LIN {X 0,Y 222.683,Z 907.794,A -85,B 0,C 180,E1 -20580.36,E2 -20580.36} C_VEL
LIN {X 0,Y 221.967,Z 912.88,A -85,B 0,C 180,E1 -20581.113,E2 -20581.113} C_VEL
LIN {X 0,Y 221.213,Z 924.782,A -85,B 0,C 180,E1 -20583.298,E2 -20583.298} C_VEL
LIN {X 0,Y 220.004,Z 934.618,A -85,B 0,C 180,E1 -20585.467,E2 -20585.467} C_VEL
LIN {X 0,Y 218.54,Z 943.393,A -85,B 0,C 180,E1 -20587.802,E2 -20587.802} C_VEL
LIN {X 0,Y 216.195,Z 951.788,A -85,B 0,C 180,E1 -20590.515,E2 -20590.515} C_VEL
LIN {X 0,Y 214.636,Z 957.677,A -85,B 0,C 180,E1 -20592.865,E2 -20592.865} C_VEL
LIN {X 0,Y 213.497,Z 963.435,A -85,B 0,C 180,E1 -20595.71,E2 -20595.71} C_VEL
LIN {X 0,Y 212.841,Z 968.001,A -85,B 0,C 180,E1 -20598.577,E2 -20598.577} C_VEL
LIN {X 0,Y 212.752,Z 972.374,A -85,B 0,C 180,E1 -20602.314,E2 -20602.314} C_VEL
LIN {X 0,Y 212.967,Z 973.999,A -85,B 0,C 180,E1 -20604.322,E2 -20604.322} C_VEL
LIN {X 0,Y 213.246,Z 975.11,A -85,B 0,C 180,E1 -20606.224,E2 -20606.224} C_VEL
LIN {X 0,Y 213.487,Z 975.797,A -85,B 0,C 180,E1 -20608.117,E2 -20608.117} C_VEL
LIN {X 0,Y 213.744,Z 976.061,A -85,B 0,C 180,E1 -20610.003,E2 -20610.003} C_VEL
LIN {X 0,Y 213.491,Z 975.785,A -85,B 0,C 180,E1 -20611.89,E2 -20611.89} C_VEL
LIN {X 0,Y 213.259,Z 975.091,A -85,B 0,C 180,E1 -20613.782,E2 -20613.782} C_VEL
LIN {X 0,Y 212.992,Z 973.972,A -85,B 0,C 180,E1 -20615.684,E2 -20615.684} C_VEL
LIN {X 0,Y 212.76,Z 972.318,A -85,B 0,C 180,E1 -20617.703,E2 -20617.703} C_VEL
LIN {X 0,Y 212.843,Z 968.742,A -85,B 0,C 180,E1 -20620.948,E2 -20620.948} C_VEL
LIN {X 0,Y 213.212,Z 967.284,A -85,B 0,C 180,E1 -20623.344,E2 -20623.344} C_VEL
LIN {X 0,Y 214.757,Z 963.862,A -85,B 0,C 180,E1 -20627.132,E2 -20627.132} C_VEL
LIN {X 0,Y 217.509,Z 959.058,A -85,B 0,C 180,E1 -20630.823,E2 -20630.823} C_VEL
LIN {X 0,Y 221.527,Z 952.942,A -85,B 0,C 180,E1 -20634.361,E2 -20634.361} C_VEL
LIN {X 0,Y 224.855,Z 947.353,A -85,B 0,C 180,E1 -20636.953,E2 -20636.953} C_VEL
LIN {X 0,Y 229.122,Z 939.872,A -85,B 0,C 180,E1 -20639.9,E2 -20639.9} C_VEL
LIN {X 0,Y 234.33,Z 930.73,A -85,B 0,C 180,E1 -20642.884,E2 -20642.884} C_VEL
LIN {X 0,Y 239.363,Z 919.685,A -85,B 0,C 180,E1 -20646.344,E2 -20646.344} C_VEL
LIN {X 0,Y 243.363,Z 909.541,A -85,B 0,C 180,E1 -20649.448,E2 -20649.448} C_VEL
LIN {X 0,Y 247.656,Z 898.848,A -85,B 0,C 180,E1 -20652.931,E2 -20652.931} C_VEL
LIN {X 0,Y 249.749,Z 893.918,A -85,B 0,C 180,E1 -20654.712,E2 -20654.712} C_VEL
LIN {X 0,Y 250.439,Z 892.26,A -85,B 0,C 180,E1 -20655.447,E2 -20655.447} C_VEL
LIN {X 0,Y 251.117,Z 890.281,A -85,B 0,C 180,E1 -20656.694,E2 -20656.694} C_VEL
LIN {X 0,Y 251.911,Z 888.053,A -85,B 0,C 180,E1 -20658.877,E2 -20658.877} C_VEL
LIN {X 0,Y 252.305,Z 887.295,A -85,B 0,C 180,E1 -20660.158,E2 -20660.158} C_VEL
LIN {X 0,Y 252.805,Z 886.985,A -85,B 0,C 180,E1 -20662.295,E2 -20662.295} C_VEL
LIN {X 0,Y 253.061,Z 887.829,A -85,B 0,C 180,E1 -20664.323,E2 -20664.323} C_VEL
LIN {X 0,Y 252.783,Z 889.741,A -85,B 0,C 180,E1 -20666.523,E2 -20666.523} C_VEL
LIN {X 0,Y 251.661,Z 893.245,A -85,B 0,C 180,E1 -20668.893,E2 -20668.893} C_VEL
LIN {X 0,Y 250.434,Z 895.146,A -85,B 0,C 180,E1 -20669.659,E2 -20669.659} C_VEL
LIN {X 0,Y 243.614,Z 903.148,A -85,B 0,C 180,E1 -20672.511,E2 -20672.511} C_VEL
LIN {X 0,Y 237.346,Z 909.214,A -85,B 0,C 180,E1 -20675.509,E2 -20675.509} C_VEL
LIN {X 0,Y 233.205,Z 912.764,A -85,B 0,C 180,E1 -20677.87,E2 -20677.87} C_VEL
LIN {X 0,Y 227.046,Z 916.649,A -85,B 0,C 180,E1 -20681.968,E2 -20681.968} C_VEL
LIN {X 0,Y 222.953,Z 918.003,A -85,B 0,C 180,E1 -20685.394,E2 -20685.394} C_VEL
LIN {X 0,Y 219.57,Z 918.045,A -85,B 0,C 180,E1 -20688.928,E2 -20688.928} C_VEL
LIN {X 0,Y 217.142,Z 916.466,A -85,B 0,C 180,E1 -20692.561,E2 -20692.561} C_VEL
LIN {X 0,Y 215.54,Z 913.407,A -85,B 0,C 180,E1 -20696.261,E2 -20696.261} C_VEL
LIN {X 0,Y 214.542,Z 910.085,A -85,B 0,C 180,E1 -20699.062,E2 -20699.062} C_VEL
LIN {X 0,Y 214.067,Z 905.794,A -85,B 0,C 180,E1 -20701.882,E2 -20701.882} C_VEL
LIN {X 0,Y 213.844,Z 899.385,A -85,B 0,C 180,E1 -20705.186,E2 -20705.186} C_VEL
LIN {X 0,Y 214.309,Z 892.64,A -85,B 0,C 180,E1 -20708.012,E2 -20708.012} C_VEL
LIN {X 0,Y 214.845,Z 884.897,A -85,B 0,C 180,E1 -20710.746,E2 -20710.746} C_VEL
LIN {X 0,Y 215.793,Z 874.678,A -85,B 0,C 180,E1 -20713.658,E2 -20713.658} C_VEL
LIN {X 0,Y 216.972,Z 862.599,A -85,B 0,C 180,E1 -20716.465,E2 -20716.465} C_VEL
LIN {X 0,Y 218.067,Z 851.603,A -85,B 0,C 180,E1 -20718.558,E2 -20718.558} C_VEL
LIN {X 0,Y 218.521,Z 845.919,A -85,B 0,C 180,E1 -20719.493,E2 -20719.493} C_VEL
LIN {X 0,Y 215.547,Z 833.553,A -85,B 0,C 180,E1 -20721.358,E2 -20721.358} C_VEL
LIN {X 0,Y 213.843,Z 825.837,A -85,B 0,C 180,E1 -20722.392,E2 -20722.392} C_VEL
LIN {X 0,Y 213.775,Z 825.841,A -85,B 0,C 180,E1 -20727.416,E2 -20727.416} C_VEL
LIN {X 0,Y 213.767,Z 825.845,A -85,B 0,C 180,E1 -20731.738,E2 -20731.738} C_VEL
LIN {X 0,Y 213.75,Z 825.853,A -85,B 0,C 180,E1 -20736.287,E2 -20736.287} C_VEL
LIN {X 0,Y 213.706,Z 825.861,A -85,B 0,C 180,E1 -20741.127,E2 -20741.127} C_VEL
LIN {X 0,Y 213.709,Z 825.861,A -85,B 0,C 180,E1 -20743.678,E2 -20743.678} C_VEL
LIN {X 0,Y 213.708,Z 825.858,A -85,B 0,C 180,E1 -20746.344,E2 -20746.344} C_VEL
LIN {X 0,Y 213.711,Z 825.865,A -85,B 0,C 180,E1 -20751.327,E2 -20751.327} C_VEL
LIN {X 0,Y 213.774,Z 825.945,A -85,B 0,C 180,E1 -20755.566,E2 -20755.566} C_VEL
LIN {X 0,Y 214.833,Z 828.734,A -85,B 0,C 180,E1 -20756.044,E2 -20756.044} C_VEL
LIN {X 0,Y 219.16,Z 837.219,A -85,B 0,C 180,E1 -20757.82,E2 -20757.82} C_VEL
LIN {X 0,Y 223.302,Z 847.04,A -85,B 0,C 180,E1 -20759.94,E2 -20759.94} C_VEL
LIN {X 0,Y 226.253,Z 856.184,A -85,B 0,C 180,E1 -20762.01,E2 -20762.01} C_VEL
LIN {X 0,Y 228.469,Z 865.319,A -85,B 0,C 180,E1 -20764.25,E2 -20764.25} C_VEL
LIN {X 0,Y 228.457,Z 867.41,A -85,B 0,C 180,E1 -20764.73,E2 -20764.73} C_VEL
LIN {X 0,Y 226.319,Z 876.166,A -85,B 0,C 180,E1 -20766.673,E2 -20766.673} C_VEL
LIN {X 0,Y 224.064,Z 884.201,A -85,B 0,C 180,E1 -20768.853,E2 -20768.853} C_VEL
LIN {X 0,Y 222.104,Z 890.846,A -85,B 0,C 180,E1 -20771.071,E2 -20771.071} C_VEL
LIN {X 0,Y 220.379,Z 896.376,A -85,B 0,C 180,E1 -20773.318,E2 -20773.318} C_VEL
LIN {X 0,Y 218.689,Z 901.747,A -85,B 0,C 180,E1 -20776.05,E2 -20776.05} C_VEL
LIN {X 0,Y 216.938,Z 906.012,A -85,B 0,C 180,E1 -20778.788,E2 -20778.788} C_VEL
LIN {X 0,Y 216.156,Z 908.239,A -85,B 0,C 180,E1 -20780.641,E2 -20780.641} C_VEL
LIN {X 0,Y 215.625,Z 910.035,A -85,B 0,C 180,E1 -20782.506,E2 -20782.506} C_VEL
LIN {X 0,Y 215.277,Z 911.377,A -85,B 0,C 180,E1 -20784.376,E2 -20784.376} C_VEL
LIN {X 0,Y 214.632,Z 912.955,A -85,B 0,C 180,E1 -20788.12,E2 -20788.12} C_VEL
LIN {X 0,Y 214.545,Z 913.183,A -85,B 0,C 180,E1 -20789.997,E2 -20789.997} C_VEL
LIN {X 0,Y 214.897,Z 912.41,A -85,B 0,C 180,E1 -20793.747,E2 -20793.747} C_VEL
LIN {X 0,Y 215.247,Z 911.466,A -85,B 0,C 180,E1 -20795.618,E2 -20795.618} C_VEL
LIN {X 0,Y 215.52,Z 910.172,A -85,B 0,C 180,E1 -20797.491,E2 -20797.491} C_VEL
LIN {X 0,Y 216.517,Z 907.366,A -85,B 0,C 180,E1 -20800.28,E2 -20800.28} C_VEL
LIN {X 0,Y 218.106,Z 903.519,A -85,B 0,C 180,E1 -20803.032,E2 -20803.032} C_VEL
LIN {X 0,Y 219.788,Z 898.601,A -85,B 0,C 180,E1 -20805.768,E2 -20805.768} C_VEL
LIN {X 0,Y 221.653,Z 892.417,A -85,B 0,C 180,E1 -20808.482,E2 -20808.482} C_VEL
LIN {X 0,Y 224.005,Z 884.641,A -85,B 0,C 180,E1 -20811.146,E2 -20811.146} C_VEL
LIN {X 0,Y 226.211,Z 876.701,A -85,B 0,C 180,E1 -20813.332,E2 -20813.332} C_VEL
LIN {X 0,Y 228.66,Z 866.99,A -85,B 0,C 180,E1 -20815.483,E2 -20815.483} C_VEL
LIN {X 0,Y 228.253,Z 863.798,A -85,B 0,C 180,E1 -20816.264,E2 -20816.264} C_VEL
LIN {X 0,Y 225.979,Z 855.105,A -85,B 0,C 180,E1 -20818.384,E2 -20818.384} C_VEL
LIN {X 0,Y 223.287,Z 846.892,A -85,B 0,C 180,E1 -20820.234,E2 -20820.234} C_VEL
LIN {X 0,Y 218.787,Z 836.479,A -85,B 0,C 180,E1 -20822.493,E2 -20822.493} C_VEL
LIN {X 0,Y 214.007,Z 826.929,A -85,B 0,C 180,E1 -20824.448,E2 -20824.448} C_VEL
LIN {X 0,Y 213.782,Z 825.857,A -85,B 0,C 180,E1 -20824.636,E2 -20824.636} C_VEL
LIN {X 0,Y 213.777,Z 825.858,A -85,B 0,C 180,E1 -20828.65,E2 -20828.65} C_VEL
LIN {X 0,Y 213.817,Z 825.851,A -85,B 0,C 180,E1 -20831.096,E2 -20831.096} C_VEL
LIN {X 0,Y 213.828,Z 825.851,A -85,B 0,C 180,E1 -20833.69,E2 -20833.69} C_VEL
LIN {X 0,Y 213.831,Z 825.846,A -85,B 0,C 180,E1 -20836.353,E2 -20836.353} C_VEL
LIN {X 0,Y 213.821,Z 825.851,A -85,B 0,C 180,E1 -20839.105,E2 -20839.105} C_VEL
LIN {X 0,Y 213.749,Z 825.859,A -85,B 0,C 180,E1 -20843.712,E2 -20843.712} C_VEL
LIN {X 0,Y 213.784,Z 825.851,A -85,B 0,C 180,E1 -20848.722,E2 -20848.722} C_VEL
LIN {X 0,Y 213.813,Z 825.852,A -85,B 0,C 180,E1 -20852.601,E2 -20852.601} C_VEL
LIN {X 0,Y 213.839,Z 825.85,A -85,B 0,C 180,E1 -20856.951,E2 -20856.951} C_VEL
LIN {X 0,Y 213.93,Z 825.834,A -85,B 0,C 180,E1 -20862.802,E2 -20862.802} C_VEL
LIN {X 0,Y 213.966,Z 825.83,A -85,B 0,C 180,E1 -20866.707,E2 -20866.707} C_VEL
LIN {X 0,Y 214.152,Z 825.8,A -85,B 0,C 180,E1 -20870.556,E2 -20870.556} C_VEL
LIN {X 0,Y 214.211,Z 825.802,A -85,B 0,C 180,E1 -20872.459,E2 -20872.459} C_VEL
LIN {X 0,Y 214.43,Z 825.773,A -85,B 0,C 180,E1 -20878.122,E2 -20878.122} C_VEL
LIN {X 0,Y 214.535,Z 825.767,A -85,B 0,C 180,E1 -20880,E2 -20880} C_VEL
LIN {X 0,Y 214.429,Z 825.78,A -85,B 0,C 180,E1 -20881.878,E2 -20881.878} C_VEL
LIN {X 0,Y 214.208,Z 825.805,A -85,B 0,C 180,E1 -20887.541,E2 -20887.541} C_VEL
LIN {X 0,Y 214.009,Z 825.822,A -85,B 0,C 180,E1 -20891.364,E2 -20891.364} C_VEL
LIN {X 0,Y 213.919,Z 825.84,A -85,B 0,C 180,E1 -20895.238,E2 -20895.238} C_VEL
LIN {X 0,Y 213.822,Z 825.853,A -85,B 0,C 180,E1 -20899.189,E2 -20899.189} C_VEL
LIN {X 0,Y 213.789,Z 825.855,A -85,B 0,C 180,E1 -20903.234,E2 -20903.234} C_VEL
LIN {X 0,Y 213.773,Z 825.851,A -85,B 0,C 180,E1 -20907.429,E2 -20907.429} C_VEL
LIN {X 0,Y 213.781,Z 826.027,A -85,B 0,C 180,E1 -20909.006,E2 -20909.006} C_VEL
LIN {X 0,Y 215.008,Z 831.466,A -85,B 0,C 180,E1 -20913.758,E2 -20913.758} C_VEL
LIN {X 0,Y 216.095,Z 836.967,A -85,B 0,C 180,E1 -20918.165,E2 -20918.165} C_VEL
LIN {X 0,Y 217.106,Z 842.018,A -85,B 0,C 180,E1 -20921.886,E2 -20921.886} C_VEL
LIN {X 0,Y 218.334,Z 848.445,A -85,B 0,C 180,E1 -20926.347,E2 -20926.347} C_VEL
LIN {X 0,Y 219.202,Z 854.278,A -85,B 0,C 180,E1 -20930.121,E2 -20930.121} C_VEL
LIN {X 0,Y 217.328,Z 861.535,A -85,B 0,C 180,E1 -20934.407,E2 -20934.407} C_VEL
LIN {X 0,Y 217.039,Z 862.617,A -85,B 0,C 180,E1 -20935.044,E2 -20935.044} C_VEL
LIN {X 0,Y 219.827,Z 877.43,A -85,B 0,C 180,E1 -20936.433,E2 -20936.433} C_VEL
LIN {X 0,Y 221.389,Z 890.305,A -85,B 0,C 180,E1 -20937.887,E2 -20937.887} C_VEL
LIN {X 0,Y 222.027,Z 903.006,A -85,B 0,C 180,E1 -20939.576,E2 -20939.576} C_VEL
LIN {X 0,Y 221.967,Z 912.88,A -85,B 0,C 180,E1 -20941.113,E2 -20941.113} C_VEL
LIN {X 0,Y 221.111,Z 917.912,A -85,B 0,C 180,E1 -20941.916,E2 -20941.916} C_VEL
LIN {X 0,Y 217.74,Z 925.844,A -85,B 0,C 180,E1 -20943.193,E2 -20943.193} C_VEL
LIN {X 0,Y 214.028,Z 933.31,A -85,B 0,C 180,E1 -20944.639,E2 -20944.639} C_VEL
LIN {X 0,Y 212.67,Z 937.55,A -85,B 0,C 180,E1 -20945.694,E2 -20945.694} C_VEL
LIN {X 0,Y 211.476,Z 943.865,A -85,B 0,C 180,E1 -20947.535,E2 -20947.535} C_VEL
LIN {X 0,Y 209.056,Z 952.07,A -85,B 0,C 180,E1 -20950.36,E2 -20950.36} C_VEL
LIN {X 0,Y 207.319,Z 958.712,A -85,B 0,C 180,E1 -20953.257,E2 -20953.257} C_VEL
LIN {X 0,Y 206.231,Z 964.049,A -85,B 0,C 180,E1 -20956.203,E2 -20956.203} C_VEL
LIN {X 0,Y 205.69,Z 968.251,A -85,B 0,C 180,E1 -20959.172,E2 -20959.172} C_VEL
LIN {X 0,Y 205.702,Z 971.488,A -85,B 0,C 180,E1 -20962.228,E2 -20962.228} C_VEL
LIN {X 0,Y 205.873,Z 972.952,A -85,B 0,C 180,E1 -20964.125,E2 -20964.125} C_VEL
LIN {X 0,Y 206.187,Z 974.072,A -85,B 0,C 180,E1 -20966.095,E2 -20966.095} C_VEL
LIN {X 0,Y 206.434,Z 974.761,A -85,B 0,C 180,E1 -20968.053,E2 -20968.053} C_VEL
LIN {X 0,Y 206.709,Z 975.028,A -85,B 0,C 180,E1 -20970.003,E2 -20970.003} C_VEL
LIN {X 0,Y 206.439,Z 974.749,A -85,B 0,C 180,E1 -20971.954,E2 -20971.954} C_VEL
LIN {X 0,Y 206.201,Z 974.052,A -85,B 0,C 180,E1 -20973.912,E2 -20973.912} C_VEL
LIN {X 0,Y 205.919,Z 972.928,A -85,B 0,C 180,E1 -20975.88,E2 -20975.88} C_VEL
LIN {X 0,Y 205.65,Z 970.404,A -85,B 0,C 180,E1 -20978.85,E2 -20978.85} C_VEL
LIN {X 0,Y 205.868,Z 967.591,A -85,B 0,C 180,E1 -20981.324,E2 -20981.324} C_VEL
LIN {X 0,Y 206.273,Z 966.276,A -85,B 0,C 180,E1 -20983.801,E2 -20983.801} C_VEL
LIN {X 0,Y 207.941,Z 963.094,A -85,B 0,C 180,E1 -20987.712,E2 -20987.712} C_VEL
LIN {X 0,Y 210.859,Z 958.713,A -85,B 0,C 180,E1 -20991.511,E2 -20991.511} C_VEL
LIN {X 0,Y 216.27,Z 951.338,A -85,B 0,C 180,E1 -20996.024,E2 -20996.024} C_VEL
LIN {X 0,Y 221.008,Z 943.837,A -85,B 0,C 180,E1 -20999.534,E2 -20999.534} C_VEL
LIN {X 0,Y 225.196,Z 937.404,A -85,B 0,C 180,E1 -21002.045,E2 -21002.045} C_VEL
LIN {X 0,Y 229.467,Z 930.54,A -85,B 0,C 180,E1 -21004.411,E2 -21004.411} C_VEL
LIN {X 0,Y 234.602,Z 920.476,A -85,B 0,C 180,E1 -21007.778,E2 -21007.778} C_VEL
LIN {X 0,Y 238.991,Z 911.214,A -85,B 0,C 180,E1 -21010.87,E2 -21010.87} C_VEL
LIN {X 0,Y 243.188,Z 902.406,A -85,B 0,C 180,E1 -21013.918,E2 -21013.918} C_VEL
LIN {X 0,Y 245.543,Z 897.892,A -85,B 0,C 180,E1 -21015.692,E2 -21015.692} C_VEL
LIN {X 0,Y 246.382,Z 895.927,A -85,B 0,C 180,E1 -21016.796,E2 -21016.796} C_VEL
LIN {X 0,Y 246.856,Z 894.714,A -85,B 0,C 180,E1 -21017.754,E2 -21017.754} C_VEL
LIN {X 0,Y 247.445,Z 893.378,A -85,B 0,C 180,E1 -21019.213,E2 -21019.213} C_VEL
LIN {X 0,Y 248.037,Z 892.425,A -85,B 0,C 180,E1 -21021.438,E2 -21021.438} C_VEL
LIN {X 0,Y 248.183,Z 892.641,A -85,B 0,C 180,E1 -21023.511,E2 -21023.511} C_VEL
LIN {X 0,Y 247.944,Z 893.919,A -85,B 0,C 180,E1 -21025.465,E2 -21025.465} C_VEL
LIN {X 0,Y 247.657,Z 894.867,A -85,B 0,C 180,E1 -21026.432,E2 -21026.432} C_VEL
LIN {X 0,Y 246.544,Z 897.179,A -85,B 0,C 180,E1 -21028.173,E2 -21028.173} C_VEL
LIN {X 0,Y 245.079,Z 899.036,A -85,B 0,C 180,E1 -21028.924,E2 -21028.924} C_VEL
LIN {X 0,Y 239.652,Z 904.776,A -85,B 0,C 180,E1 -21031.061,E2 -21031.061} C_VEL
LIN {X 0,Y 232.928,Z 910.767,A -85,B 0,C 180,E1 -21034.056,E2 -21034.056} C_VEL
LIN {X 0,Y 228.423,Z 914.285,A -85,B 0,C 180,E1 -21036.423,E2 -21036.423} C_VEL
LIN {X 0,Y 225.661,Z 916.099,A -85,B 0,C 180,E1 -21038.054,E2 -21038.054} C_VEL
LIN {X 0,Y 220.57,Z 918.549,A -85,B 0,C 180,E1 -21041.42,E2 -21041.42} C_VEL
LIN {X 0,Y 218.324,Z 919.318,A -85,B 0,C 180,E1 -21043.159,E2 -21043.159} C_VEL
LIN {X 0,Y 214.415,Z 919.665,A -85,B 0,C 180,E1 -21046.736,E2 -21046.736} C_VEL
LIN {X 0,Y 212.716,Z 919.295,A -85,B 0,C 180,E1 -21048.566,E2 -21048.566} C_VEL
LIN {X 0,Y 210.19,Z 917.429,A -85,B 0,C 180,E1 -21052.314,E2 -21052.314} C_VEL
LIN {X 0,Y 208.477,Z 913.961,A -85,B 0,C 180,E1 -21056.134,E2 -21056.134} C_VEL
LIN {X 0,Y 207.445,Z 910.398,A -85,B 0,C 180,E1 -21059.029,E2 -21059.029} C_VEL
LIN {X 0,Y 206.964,Z 905.852,A -85,B 0,C 180,E1 -21061.946,E2 -21061.946} C_VEL
LIN {X 0,Y 206.738,Z 900.23,A -85,B 0,C 180,E1 -21064.875,E2 -21064.875} C_VEL
LIN {X 0,Y 207.156,Z 893.416,A -85,B 0,C 180,E1 -21067.799,E2 -21067.799} C_VEL
LIN {X 0,Y 207.657,Z 886.611,A -85,B 0,C 180,E1 -21070.291,E2 -21070.291} C_VEL
LIN {X 0,Y 208.354,Z 878.805,A -85,B 0,C 180,E1 -21072.665,E2 -21072.665} C_VEL
LIN {X 0,Y 209.142,Z 870.512,A -85,B 0,C 180,E1 -21074.847,E2 -21074.847} C_VEL
LIN {X 0,Y 209.99,Z 861.955,A -85,B 0,C 180,E1 -21076.778,E2 -21076.778} C_VEL
LIN {X 0,Y 211.155,Z 850.698,A -85,B 0,C 180,E1 -21078.936,E2 -21078.936} C_VEL
LIN {X 0,Y 211.291,Z 846.213,A -85,B 0,C 180,E1 -21079.687,E2 -21079.687} C_VEL
LIN {X 0,Y 208.404,Z 834.211,A -85,B 0,C 180,E1 -21081.54,E2 -21081.54} C_VEL
LIN {X 0,Y 206.788,Z 826.717,A -85,B 0,C 180,E1 -21082.571,E2 -21082.571} C_VEL
LIN {X 0,Y 206.704,Z 826.722,A -85,B 0,C 180,E1 -21087.865,E2 -21087.865} C_VEL
LIN {X 0,Y 206.717,Z 826.723,A -85,B 0,C 180,E1 -21091.788,E2 -21091.788} C_VEL
LIN {X 0,Y 206.708,Z 826.733,A -85,B 0,C 180,E1 -21095.31,E2 -21095.31} C_VEL
LIN {X 0,Y 206.655,Z 826.742,A -85,B 0,C 180,E1 -21100.253,E2 -21100.253} C_VEL
LIN {X 0,Y 206.637,Z 826.746,A -85,B 0,C 180,E1 -21104.415,E2 -21104.415} C_VEL
LIN {X 0,Y 206.637,Z 826.746,A -85,B 0,C 180,E1 -21108.439,E2 -21108.439} C_VEL
LIN {X 0,Y 206.698,Z 826.733,A -85,B 0,C 180,E1 -21113.483,E2 -21113.483} C_VEL
LIN {X 0,Y 206.736,Z 826.85,A -85,B 0,C 180,E1 -21114.18,E2 -21114.18} C_VEL
LIN {X 0,Y 207.778,Z 829.656,A -85,B 0,C 180,E1 -21114.689,E2 -21114.689} C_VEL
LIN {X 0,Y 212.372,Z 838.462,A -85,B 0,C 180,E1 -21116.667,E2 -21116.667} C_VEL
LIN {X 0,Y 216.471,Z 848.029,A -85,B 0,C 180,E1 -21118.858,E2 -21118.858} C_VEL
LIN {X 0,Y 219.657,Z 857.627,A -85,B 0,C 180,E1 -21121.156,E2 -21121.156} C_VEL
LIN {X 0,Y 221.764,Z 866.251,A -85,B 0,C 180,E1 -21123.373,E2 -21123.373} C_VEL
LIN {X 0,Y 222.115,Z 868.447,A -85,B 0,C 180,E1 -21123.955,E2 -21123.955} C_VEL
LIN {X 0,Y 219.887,Z 877.2,A -85,B 0,C 180,E1 -21125.948,E2 -21125.948} C_VEL
LIN {X 0,Y 217.527,Z 885.234,A -85,B 0,C 180,E1 -21128.186,E2 -21128.186} C_VEL
LIN {X 0,Y 215.47,Z 891.879,A -85,B 0,C 180,E1 -21130.465,E2 -21130.465} C_VEL
LIN {X 0,Y 213.659,Z 897.409,A -85,B 0,C 180,E1 -21132.777,E2 -21132.777} C_VEL
LIN {X 0,Y 211.88,Z 902.78,A -85,B 0,C 180,E1 -21135.592,E2 -21135.592} C_VEL
LIN {X 0,Y 210.053,Z 907.044,A -85,B 0,C 180,E1 -21138.416,E2 -21138.416} C_VEL
LIN {X 0,Y 209.228,Z 909.271,A -85,B 0,C 180,E1 -21140.328,E2 -21140.328} C_VEL
LIN {X 0,Y 208.673,Z 911.066,A -85,B 0,C 180,E1 -21142.254,E2 -21142.254} C_VEL
LIN {X 0,Y 208.291,Z 912.408,A -85,B 0,C 180,E1 -21144.187,E2 -21144.187} C_VEL
LIN {X 0,Y 207.612,Z 913.986,A -85,B 0,C 180,E1 -21148.057,E2 -21148.057} C_VEL
LIN {X 0,Y 207.521,Z 914.214,A -85,B 0,C 180,E1 -21149.997,E2 -21149.997} C_VEL
LIN {X 0,Y 207.888,Z 913.441,A -85,B 0,C 180,E1 -21153.873,E2 -21153.873} C_VEL
LIN {X 0,Y 208.258,Z 912.496,A -85,B 0,C 180,E1 -21155.807,E2 -21155.807} C_VEL
LIN {X 0,Y 208.581,Z 911.199,A -85,B 0,C 180,E1 -21157.742,E2 -21157.742} C_VEL
LIN {X 0,Y 209.609,Z 908.397,A -85,B 0,C 180,E1 -21160.623,E2 -21160.623} C_VEL
LIN {X 0,Y 211.267,Z 904.549,A -85,B 0,C 180,E1 -21163.462,E2 -21163.462} C_VEL
LIN {X 0,Y 213.036,Z 899.631,A -85,B 0,C 180,E1 -21166.281,E2 -21166.281} C_VEL
LIN {X 0,Y 215.009,Z 893.445,A -85,B 0,C 180,E1 -21169.075,E2 -21169.075} C_VEL
LIN {X 0,Y 217.469,Z 885.67,A -85,B 0,C 180,E1 -21171.813,E2 -21171.813} C_VEL
LIN {X 0,Y 219.779,Z 877.73,A -85,B 0,C 180,E1 -21174.057,E2 -21174.057} C_VEL
LIN {X 0,Y 222.226,Z 868.036,A -85,B 0,C 180,E1 -21176.276,E2 -21176.276} C_VEL
LIN {X 0,Y 220.133,Z 859.17,A -85,B 0,C 180,E1 -21178.609,E2 -21178.609} C_VEL
LIN {X 0,Y 217.112,Z 849.564,A -85,B 0,C 180,E1 -21180.929,E2 -21180.929} C_VEL
LIN {X 0,Y 212.971,Z 839.724,A -85,B 0,C 180,E1 -21183.205,E2 -21183.205} C_VEL
LIN {X 0,Y 208.128,Z 830.196,A -85,B 0,C 180,E1 -21185.343,E2 -21185.343} C_VEL
LIN {X 0,Y 206.858,Z 827.511,A -85,B 0,C 180,E1 -21185.888,E2 -21185.888} C_VEL
LIN {X 0,Y 206.708,Z 826.738,A -85,B 0,C 180,E1 -21186.039,E2 -21186.039} C_VEL
LIN {X 0,Y 206.736,Z 826.736,A -85,B 0,C 180,E1 -21190.228,E2 -21190.228} C_VEL
LIN {X 0,Y 206.737,Z 826.733,A -85,B 0,C 180,E1 -21194.447,E2 -21194.447} C_VEL
LIN {X 0,Y 206.744,Z 826.728,A -85,B 0,C 180,E1 -21198.399,E2 -21198.399} C_VEL
LIN {X 0,Y 206.735,Z 826.727,A -85,B 0,C 180,E1 -21202.272,E2 -21202.272} C_VEL
LIN {X 0,Y 206.698,Z 826.736,A -85,B 0,C 180,E1 -21207.042,E2 -21207.042} C_VEL
LIN {X 0,Y 206.754,Z 826.73,A -85,B 0,C 180,E1 -21212.094,E2 -21212.094} C_VEL
LIN {X 0,Y 206.772,Z 826.728,A -85,B 0,C 180,E1 -21216.582,E2 -21216.582} C_VEL
LIN {X 0,Y 206.86,Z 826.717,A -85,B 0,C 180,E1 -21222.195,E2 -21222.195} C_VEL
LIN {X 0,Y 206.9,Z 826.708,A -85,B 0,C 180,E1 -21226.244,E2 -21226.244} C_VEL
LIN {X 0,Y 207.091,Z 826.68,A -85,B 0,C 180,E1 -21230.23,E2 -21230.23} C_VEL
LIN {X 0,Y 207.152,Z 826.678,A -85,B 0,C 180,E1 -21232.2,E2 -21232.2} C_VEL
LIN {X 0,Y 207.367,Z 826.652,A -85,B 0,C 180,E1 -21238.058,E2 -21238.058} C_VEL
LIN {X 0,Y 207.5,Z 826.644,A -85,B 0,C 180,E1 -21240,E2 -21240} C_VEL
LIN {X 0,Y 207.365,Z 826.66,A -85,B 0,C 180,E1 -21241.942,E2 -21241.942} C_VEL
LIN {X 0,Y 207.149,Z 826.684,A -85,B 0,C 180,E1 -21247.8,E2 -21247.8} C_VEL
LIN {X 0,Y 206.929,Z 826.7,A -85,B 0,C 180,E1 -21251.758,E2 -21251.758} C_VEL
LIN {X 0,Y 206.853,Z 826.719,A -85,B 0,C 180,E1 -21255.772,E2 -21255.772} C_VEL
LIN {X 0,Y 206.765,Z 826.731,A -85,B 0,C 180,E1 -21259.871,E2 -21259.871} C_VEL
LIN {X 0,Y 206.724,Z 826.736,A -85,B 0,C 180,E1 -21264.077,E2 -21264.077} C_VEL
LIN {X 0,Y 206.723,Z 826.776,A -85,B 0,C 180,E1 -21267.696,E2 -21267.696} C_VEL
LIN {X 0,Y 207.926,Z 832.213,A -85,B 0,C 180,E1 -21272.739,E2 -21272.739} C_VEL
LIN {X 0,Y 209.008,Z 837.586,A -85,B 0,C 180,E1 -21277.248,E2 -21277.248} C_VEL
LIN {X 0,Y 210.227,Z 843.74,A -85,B 0,C 180,E1 -21281.96,E2 -21281.96} C_VEL
LIN {X 0,Y 211.2,Z 848.895,A -85,B 0,C 180,E1 -21285.674,E2 -21285.674} C_VEL
LIN {X 0,Y 212.13,Z 854.733,A -85,B 0,C 180,E1 -21289.641,E2 -21289.641} C_VEL
LIN {X 0,Y 211.317,Z 858.595,A -85,B 0,C 180,E1 -21292.033,E2 -21292.033} C_VEL
LIN {X 0,Y 210.511,Z 861.47,A -85,B 0,C 180,E1 -21293.784,E2 -21293.784} C_VEL
LIN {X 0,Y 211.912,Z 868.599,A -85,B 0,C 180,E1 -21294.457,E2 -21294.457} C_VEL
LIN {X 0,Y 214.185,Z 882.275,A -85,B 0,C 180,E1 -21295.947,E2 -21295.947} C_VEL
LIN {X 0,Y 215.257,Z 894.89,A -85,B 0,C 180,E1 -21297.543,E2 -21297.543} C_VEL
LIN {X 0,Y 215.488,Z 907.149,A -85,B 0,C 180,E1 -21299.367,E2 -21299.367} C_VEL
LIN {X 0,Y 215.002,Z 918.657,A -85,B 0,C 180,E1 -21301.395,E2 -21301.395} C_VEL
LIN {X 0,Y 214.023,Z 928.405,A -85,B 0,C 180,E1 -21303.426,E2 -21303.426} C_VEL
LIN {X 0,Y 212.67,Z 937.55,A -85,B 0,C 180,E1 -21305.694,E2 -21305.694} C_VEL
LIN {X 0,Y 211.17,Z 941.647,A -85,B 0,C 180,E1 -21306.8,E2 -21306.8} C_VEL
LIN {X 0,Y 208.654,Z 945.396,A -85,B 0,C 180,E1 -21307.87,E2 -21307.87} C_VEL
LIN {X 0,Y 203.024,Z 952.082,A -85,B 0,C 180,E1 -21310.149,E2 -21310.149} C_VEL
LIN {X 0,Y 201.114,Z 955.188,A -85,B 0,C 180,E1 -21311.476,E2 -21311.476} C_VEL
LIN {X 0,Y 200.78,Z 956.183,A -85,B 0,C 180,E1 -21311.95,E2 -21311.95} C_VEL
LIN {X 0,Y 199.64,Z 961.334,A -85,B 0,C 180,E1 -21314.695,E2 -21314.695} C_VEL
LIN {X 0,Y 198.823,Z 965.9,A -85,B 0,C 180,E1 -21317.759,E2 -21317.759} C_VEL
LIN {X 0,Y 198.58,Z 969.403,A -85,B 0,C 180,E1 -21320.84,E2 -21320.84} C_VEL
LIN {X 0,Y 198.785,Z 971.906,A -85,B 0,C 180,E1 -21323.915,E2 -21323.915} C_VEL
LIN {X 0,Y 199.125,Z 973.033,A -85,B 0,C 180,E1 -21325.956,E2 -21325.956} C_VEL
LIN {X 0,Y 199.38,Z 973.725,A -85,B 0,C 180,E1 -21327.984,E2 -21327.984} C_VEL
LIN {X 0,Y 199.672,Z 973.995,A -85,B 0,C 180,E1 -21330.004,E2 -21330.004} C_VEL
LIN {X 0,Y 199.386,Z 973.713,A -85,B 0,C 180,E1 -21332.024,E2 -21332.024} C_VEL
LIN {X 0,Y 199.142,Z 973.013,A -85,B 0,C 180,E1 -21334.051,E2 -21334.051} C_VEL
LIN {X 0,Y 198.655,Z 970.549,A -85,B 0,C 180,E1 -21337.87,E2 -21337.87} C_VEL
LIN {X 0,Y 198.951,Z 966.151,A -85,B 0,C 180,E1 -21342.24,E2 -21342.24} C_VEL
LIN {X 0,Y 200.111,Z 963.966,A -85,B 0,C 180,E1 -21346.321,E2 -21346.321} C_VEL
LIN {X 0,Y 202.695,Z 960.231,A -85,B 0,C 180,E1 -21350.583,E2 -21350.583} C_VEL
LIN {X 0,Y 206.289,Z 955.813,A -85,B 0,C 180,E1 -21354.134,E2 -21354.134} C_VEL
LIN {X 0,Y 211.071,Z 949.827,A -85,B 0,C 180,E1 -21357.788,E2 -21357.788} C_VEL
LIN {X 0,Y 216.251,Z 942.522,A -85,B 0,C 180,E1 -21361.335,E2 -21361.335} C_VEL
LIN {X 0,Y 221.742,Z 935.05,A -85,B 0,C 180,E1 -21364.276,E2 -21364.276} C_VEL
LIN {X 0,Y 226.677,Z 927.104,A -85,B 0,C 180,E1 -21367.202,E2 -21367.202} C_VEL
LIN {X 0,Y 232.653,Z 916.593,A -85,B 0,C 180,E1 -21370.957,E2 -21370.957} C_VEL
LIN {X 0,Y 238.323,Z 906.498,A -85,B 0,C 180,E1 -21374.69,E2 -21374.69} C_VEL
LIN {X 0,Y 240.009,Z 903.601,A -85,B 0,C 180,E1 -21375.808,E2 -21375.808} C_VEL
LIN {X 0,Y 241.113,Z 901.604,A -85,B 0,C 180,E1 -21376.781,E2 -21376.781} C_VEL
LIN {X 0,Y 242.032,Z 899.742,A -85,B 0,C 180,E1 -21378.098,E2 -21378.098} C_VEL
LIN {X 0,Y 242.907,Z 897.934,A -85,B 0,C 180,E1 -21380.467,E2 -21380.467} C_VEL
LIN {X 0,Y 243.255,Z 897.591,A -85,B 0,C 180,E1 -21382.647,E2 -21382.647} C_VEL
LIN {X 0,Y 242.948,Z 898.391,A -85,B 0,C 180,E1 -21384.651,E2 -21384.651} C_VEL
LIN {X 0,Y 242.108,Z 899.984,A -85,B 0,C 180,E1 -21386.527,E2 -21386.527} C_VEL
LIN {X 0,Y 241.446,Z 901.058,A -85,B 0,C 180,E1 -21387.419,E2 -21387.419} C_VEL
LIN {X 0,Y 234.037,Z 908.082,A -85,B 0,C 180,E1 -21390.298,E2 -21390.298} C_VEL
LIN {X 0,Y 228.716,Z 912.411,A -85,B 0,C 180,E1 -21392.553,E2 -21392.553} C_VEL
LIN {X 0,Y 225.444,Z 914.853,A -85,B 0,C 180,E1 -21394.123,E2 -21394.123} C_VEL
LIN {X 0,Y 219.408,Z 918.345,A -85,B 0,C 180,E1 -21397.395,E2 -21397.395} C_VEL
LIN {X 0,Y 216.683,Z 919.648,A -85,B 0,C 180,E1 -21399.097,E2 -21399.097} C_VEL
LIN {X 0,Y 211.752,Z 921.027,A -85,B 0,C 180,E1 -21402.62,E2 -21402.62} C_VEL
LIN {X 0,Y 207.654,Z 921.047,A -85,B 0,C 180,E1 -21406.296,E2 -21406.296} C_VEL
LIN {X 0,Y 205.882,Z 920.519,A -85,B 0,C 180,E1 -21408.181,E2 -21408.181} C_VEL
LIN {X 0,Y 204.516,Z 919.563,A -85,B 0,C 180,E1 -21410.106,E2 -21410.106} C_VEL
LIN {X 0,Y 202.269,Z 916.584,A -85,B 0,C 180,E1 -21414.017,E2 -21414.017} C_VEL
LIN {X 0,Y 200.73,Z 912.078,A -85,B 0,C 180,E1 -21417.994,E2 -21417.994} C_VEL
LIN {X 0,Y 199.986,Z 907.613,A -85,B 0,C 180,E1 -21421.007,E2 -21421.007} C_VEL
LIN {X 0,Y 199.642,Z 901.019,A -85,B 0,C 180,E1 -21424.543,E2 -21424.543} C_VEL
LIN {X 0,Y 199.897,Z 895.387,A -85,B 0,C 180,E1 -21427.068,E2 -21427.068} C_VEL
LIN {X 0,Y 200.527,Z 887.438,A -85,B 0,C 180,E1 -21430.093,E2 -21430.093} C_VEL
LIN {X 0,Y 201.224,Z 879.372,A -85,B 0,C 180,E1 -21432.609,E2 -21432.609} C_VEL
LIN {X 0,Y 202.119,Z 870.001,A -85,B 0,C 180,E1 -21435.117,E2 -21435.117} C_VEL
LIN {X 0,Y 203.259,Z 858.878,A -85,B 0,C 180,E1 -21437.611,E2 -21437.611} C_VEL
LIN {X 0,Y 204.336,Z 848.166,A -85,B 0,C 180,E1 -21439.594,E2 -21439.594} C_VEL
LIN {X 0,Y 201.555,Z 836.057,A -85,B 0,C 180,E1 -21441.542,E2 -21441.542} C_VEL
LIN {X 0,Y 199.751,Z 827.595,A -85,B 0,C 180,E1 -21442.77,E2 -21442.77} C_VEL
LIN {X 0,Y 199.664,Z 827.602,A -85,B 0,C 180,E1 -21448.354,E2 -21448.354} C_VEL
LIN {X 0,Y 199.673,Z 827.597,A -85,B 0,C 180,E1 -21452.351,E2 -21452.351} C_VEL
LIN {X 0,Y 199.625,Z 827.609,A -85,B 0,C 180,E1 -21456.763,E2 -21456.763} C_VEL
LIN {X 0,Y 199.602,Z 827.617,A -85,B 0,C 180,E1 -21459.33,E2 -21459.33} C_VEL
LIN {X 0,Y 199.573,Z 827.615,A -85,B 0,C 180,E1 -21462.305,E2 -21462.305} C_VEL
LIN {X 0,Y 199.583,Z 827.621,A -85,B 0,C 180,E1 -21465.225,E2 -21465.225} C_VEL
LIN {X 0,Y 199.577,Z 827.626,A -85,B 0,C 180,E1 -21468,E2 -21468} C_VEL
LIN {X 0,Y 199.658,Z 827.772,A -85,B 0,C 180,E1 -21472.661,E2 -21472.661} C_VEL
LIN {X 0,Y 200.723,Z 830.562,A -85,B 0,C 180,E1 -21473.208,E2 -21473.208} C_VEL
LIN {X 0,Y 205.3,Z 838.893,A -85,B 0,C 180,E1 -21475.245,E2 -21475.245} C_VEL
LIN {X 0,Y 209.78,Z 849.322,A -85,B 0,C 180,E1 -21477.769,E2 -21477.769} C_VEL
LIN {X 0,Y 212.896,Z 858.333,A -85,B 0,C 180,E1 -21480.061,E2 -21480.061} C_VEL
LIN {X 0,Y 215.082,Z 867.211,A -85,B 0,C 180,E1 -21482.442,E2 -21482.442} C_VEL
LIN {X 0,Y 215.54,Z 870.532,A -85,B 0,C 180,E1 -21483.36,E2 -21483.36} C_VEL
LIN {X 0,Y 213.494,Z 878.234,A -85,B 0,C 180,E1 -21485.18,E2 -21485.18} C_VEL
LIN {X 0,Y 211.022,Z 886.268,A -85,B 0,C 180,E1 -21487.477,E2 -21487.477} C_VEL
LIN {X 0,Y 208.861,Z 892.913,A -85,B 0,C 180,E1 -21489.821,E2 -21489.821} C_VEL
LIN {X 0,Y 206.976,Z 898.439,A -85,B 0,C 180,E1 -21492.202,E2 -21492.202} C_VEL
LIN {X 0,Y 205.084,Z 903.812,A -85,B 0,C 180,E1 -21495.104,E2 -21495.104} C_VEL
LIN {X 0,Y 203.177,Z 908.076,A -85,B 0,C 180,E1 -21498.018,E2 -21498.018} C_VEL
LIN {X 0,Y 202.306,Z 910.303,A -85,B 0,C 180,E1 -21499.994,E2 -21499.994} C_VEL
LIN {X 0,Y 201.723,Z 912.096,A -85,B 0,C 180,E1 -21501.986,E2 -21501.986} C_VEL
LIN {X 0,Y 201.308,Z 913.439,A -85,B 0,C 180,E1 -21503.985,E2 -21503.985} C_VEL
LIN {X 0,Y 200.592,Z 915.018,A -85,B 0,C 180,E1 -21507.989,E2 -21507.989} C_VEL
LIN {X 0,Y 200.497,Z 915.245,A -85,B 0,C 180,E1 -21509.996,E2 -21509.996} C_VEL
LIN {X 0,Y 200.881,Z 914.472,A -85,B 0,C 180,E1 -21514.009,E2 -21514.009} C_VEL
LIN {X 0,Y 201.273,Z 913.527,A -85,B 0,C 180,E1 -21516.009,E2 -21516.009} C_VEL
LIN {X 0,Y 201.642,Z 912.227,A -85,B 0,C 180,E1 -21518.01,E2 -21518.01} C_VEL
LIN {X 0,Y 202.708,Z 909.427,A -85,B 0,C 180,E1 -21520.989,E2 -21520.989} C_VEL
LIN {X 0,Y 204.441,Z 905.579,A -85,B 0,C 180,E1 -21523.92,E2 -21523.92} C_VEL
LIN {X 0,Y 206.302,Z 900.66,A -85,B 0,C 180,E1 -21526.828,E2 -21526.828} C_VEL
LIN {X 0,Y 208.385,Z 894.474,A -85,B 0,C 180,E1 -21529.706,E2 -21529.706} C_VEL
LIN {X 0,Y 210.963,Z 886.699,A -85,B 0,C 180,E1 -21532.522,E2 -21532.522} C_VEL
LIN {X 0,Y 213.385,Z 878.758,A -85,B 0,C 180,E1 -21534.826,E2 -21534.826} C_VEL
LIN {X 0,Y 215.75,Z 870.1,A -85,B 0,C 180,E1 -21536.866,E2 -21536.866} C_VEL
LIN {X 0,Y 213.758,Z 861.457,A -85,B 0,C 180,E1 -21539.276,E2 -21539.276} C_VEL
LIN {X 0,Y 211.171,Z 852.9,A -85,B 0,C 180,E1 -21541.48,E2 -21541.48} C_VEL
LIN {X 0,Y 206.727,Z 842.015,A -85,B 0,C 180,E1 -21544.181,E2 -21544.181} C_VEL
LIN {X 0,Y 201.52,Z 831.574,A -85,B 0,C 180,E1 -21546.666,E2 -21546.666} C_VEL
LIN {X 0,Y 200.007,Z 829.054,A -85,B 0,C 180,E1 -21547.289,E2 -21547.289} C_VEL
LIN {X 0,Y 199.678,Z 827.614,A -85,B 0,C 180,E1 -21547.557,E2 -21547.557} C_VEL
LIN {X 0,Y 199.682,Z 827.613,A -85,B 0,C 180,E1 -21552.344,E2 -21552.344} C_VEL
LIN {X 0,Y 199.685,Z 827.612,A -85,B 0,C 180,E1 -21555.258,E2 -21555.258} C_VEL
LIN {X 0,Y 199.687,Z 827.604,A -85,B 0,C 180,E1 -21558.032,E2 -21558.032} C_VEL
LIN {X 0,Y 199.715,Z 827.601,A -85,B 0,C 180,E1 -21560.724,E2 -21560.724} C_VEL
LIN {X 0,Y 199.623,Z 827.61,A -85,B 0,C 180,E1 -21565.715,E2 -21565.715} C_VEL
LIN {X 0,Y 199.692,Z 827.611,A -85,B 0,C 180,E1 -21568.135,E2 -21568.135} C_VEL
LIN {X 0,Y 199.675,Z 827.612,A -85,B 0,C 180,E1 -21572.77,E2 -21572.77} C_VEL
LIN {X 0,Y 199.725,Z 827.606,A -85,B 0,C 180,E1 -21577.227,E2 -21577.227} C_VEL
LIN {X 0,Y 199.783,Z 827.599,A -85,B 0,C 180,E1 -21581.756,E2 -21581.756} C_VEL
LIN {X 0,Y 199.834,Z 827.583,A -85,B 0,C 180,E1 -21585.748,E2 -21585.748} C_VEL
LIN {X 0,Y 200.056,Z 827.558,A -85,B 0,C 180,E1 -21589.883,E2 -21589.883} C_VEL
LIN {X 0,Y 200.019,Z 827.576,A -85,B 0,C 180,E1 -21593.949,E2 -21593.949} C_VEL
LIN {X 0,Y 200.306,Z 827.531,A -85,B 0,C 180,E1 -21597.989,E2 -21597.989} C_VEL
LIN {X 0,Y 200.464,Z 827.52,A -85,B 0,C 180,E1 -21600,E2 -21600} C_VEL
LIN {X 0,Y 200.011,Z 827.573,A -85,B 0,C 180,E1 -21604.03,E2 -21604.03} C_VEL
LIN {X 0,Y 200.094,Z 827.561,A -85,B 0,C 180,E1 -21608.076,E2 -21608.076} C_VEL
LIN {X 0,Y 200.022,Z 827.57,A -85,B 0,C 180,E1 -21610.348,E2 -21610.348} C_VEL
LIN {X 0,Y 199.79,Z 827.6,A -85,B 0,C 180,E1 -21616.345,E2 -21616.345} C_VEL
LIN {X 0,Y 199.676,Z 827.616,A -85,B 0,C 180,E1 -21620.608,E2 -21620.608} C_VEL
LIN {X 0,Y 199.637,Z 827.617,A -85,B 0,C 180,E1 -21624.989,E2 -21624.989} C_VEL
LIN {X 0,Y 199.655,Z 827.621,A -85,B 0,C 180,E1 -21626.386,E2 -21626.386} C_VEL
LIN {X 0,Y 200.565,Z 831.795,A -85,B 0,C 180,E1 -21630.537,E2 -21630.537} C_VEL
LIN {X 0,Y 201.672,Z 836.84,A -85,B 0,C 180,E1 -21635.1,E2 -21635.1} C_VEL
LIN {X 0,Y 202.893,Z 843.238,A -85,B 0,C 180,E1 -21640.361,E2 -21640.361} C_VEL
LIN {X 0,Y 204.062,Z 849.259,A -85,B 0,C 180,E1 -21644.913,E2 -21644.913} C_VEL
LIN {X 0,Y 205.022,Z 854.923,A -85,B 0,C 180,E1 -21648.951,E2 -21648.951} C_VEL
LIN {X 0,Y 204.82,Z 857.42,A -85,B 0,C 180,E1 -21650.601,E2 -21650.601} C_VEL
LIN {X 0,Y 204.019,Z 860.326,A -85,B 0,C 180,E1 -21652.441,E2 -21652.441} C_VEL
LIN {X 0,Y 206.873,Z 875.549,A -85,B 0,C 180,E1 -21654.052,E2 -21654.052} C_VEL
LIN {X 0,Y 208.474,Z 888.465,A -85,B 0,C 180,E1 -21655.682,E2 -21655.682} C_VEL
LIN {X 0,Y 209.003,Z 900.776,A -85,B 0,C 180,E1 -21657.456,E2 -21657.456} C_VEL
LIN {X 0,Y 208.828,Z 912.373,A -85,B 0,C 180,E1 -21659.423,E2 -21659.423} C_VEL
LIN {X 0,Y 207.911,Z 923.991,A -85,B 0,C 180,E1 -21661.76,E2 -21661.76} C_VEL
LIN {X 0,Y 206.383,Z 934.329,A -85,B 0,C 180,E1 -21664.271,E2 -21664.271} C_VEL
LIN {X 0,Y 204.852,Z 942.812,A -85,B 0,C 180,E1 -21666.767,E2 -21666.767} C_VEL
LIN {X 0,Y 202.386,Z 951.03,A -85,B 0,C 180,E1 -21669.684,E2 -21669.684} C_VEL
LIN {X 0,Y 200.78,Z 956.183,A -85,B 0,C 180,E1 -21671.95,E2 -21671.95} C_VEL
LIN {X 0,Y 199.449,Z 959.04,A -85,B 0,C 180,E1 -21673.387,E2 -21673.387} C_VEL
LIN {X 0,Y 195.701,Z 962.974,A -85,B 0,C 180,E1 -21675.798,E2 -21675.798} C_VEL
LIN {X 0,Y 192.824,Z 965.604,A -85,B 0,C 180,E1 -21677.849,E2 -21677.849} C_VEL
LIN {X 0,Y 191.621,Z 967.378,A -85,B 0,C 180,E1 -21679.496,E2 -21679.496} C_VEL
LIN {X 0,Y 191.525,Z 967.922,A -85,B 0,C 180,E1 -21680.061,E2 -21680.061} C_VEL
LIN {X 0,Y 191.699,Z 970.86,A -85,B 0,C 180,E1 -21683.689,E2 -21683.689} C_VEL
LIN {X 0,Y 192.061,Z 971.994,A -85,B 0,C 180,E1 -21685.807,E2 -21685.807} C_VEL
LIN {X 0,Y 192.324,Z 972.688,A -85,B 0,C 180,E1 -21687.91,E2 -21687.91} C_VEL
LIN {X 0,Y 192.633,Z 972.961,A -85,B 0,C 180,E1 -21690.004,E2 -21690.004} C_VEL
LIN {X 0,Y 192.331,Z 972.676,A -85,B 0,C 180,E1 -21692.098,E2 -21692.098} C_VEL
LIN {X 0,Y 192.08,Z 971.973,A -85,B 0,C 180,E1 -21694.2,E2 -21694.2} C_VEL
LIN {X 0,Y 191.584,Z 969.682,A -85,B 0,C 180,E1 -21697.921,E2 -21697.921} C_VEL
LIN {X 0,Y 191.876,Z 965.469,A -85,B 0,C 180,E1 -21702.162,E2 -21702.162} C_VEL
LIN {X 0,Y 192.008,Z 964.895,A -85,B 0,C 180,E1 -21702.69,E2 -21702.69} C_VEL
LIN {X 0,Y 193.28,Z 962.984,A -85,B 0,C 180,E1 -21706.915,E2 -21706.915} C_VEL
LIN {X 0,Y 195.846,Z 959.745,A -85,B 0,C 180,E1 -21711.089,E2 -21711.089} C_VEL
LIN {X 0,Y 199.799,Z 955.492,A -85,B 0,C 180,E1 -21714.971,E2 -21714.971} C_VEL
LIN {X 0,Y 204.787,Z 949.968,A -85,B 0,C 180,E1 -21718.719,E2 -21718.719} C_VEL
LIN {X 0,Y 210.249,Z 943.253,A -85,B 0,C 180,E1 -21722.336,E2 -21722.336} C_VEL
LIN {X 0,Y 217.437,Z 934.345,A -85,B 0,C 180,E1 -21726.094,E2 -21726.094} C_VEL
LIN {X 0,Y 224.144,Z 924.368,A -85,B 0,C 180,E1 -21730.003,E2 -21730.003} C_VEL
LIN {X 0,Y 229.936,Z 915.472,A -85,B 0,C 180,E1 -21733.453,E2 -21733.453} C_VEL
LIN {X 0,Y 235.087,Z 907.785,A -85,B 0,C 180,E1 -21736.56,E2 -21736.56} C_VEL
LIN {X 0,Y 236.634,Z 905.323,A -85,B 0,C 180,E1 -21737.948,E2 -21737.948} C_VEL
LIN {X 0,Y 237.463,Z 903.784,A -85,B 0,C 180,E1 -21739.374,E2 -21739.374} C_VEL
LIN {X 0,Y 238.073,Z 902.612,A -85,B 0,C 180,E1 -21741.689,E2 -21741.689} C_VEL
LIN {X 0,Y 238.074,Z 902.594,A -85,B 0,C 180,E1 -21742.853,E2 -21742.853} C_VEL
LIN {X 0,Y 237.879,Z 902.824,A -85,B 0,C 180,E1 -21743.78,E2 -21743.78} C_VEL
LIN {X 0,Y 236.584,Z 904.476,A -85,B 0,C 180,E1 -21746.285,E2 -21746.285} C_VEL
LIN {X 0,Y 235.687,Z 905.353,A -85,B 0,C 180,E1 -21746.841,E2 -21746.841} C_VEL
LIN {X 0,Y 230.381,Z 909.907,A -85,B 0,C 180,E1 -21748.761,E2 -21748.761} C_VEL
LIN {X 0,Y 224.737,Z 914.132,A -85,B 0,C 180,E1 -21751.006,E2 -21751.006} C_VEL
LIN {X 0,Y 219.512,Z 917.534,A -85,B 0,C 180,E1 -21753.37,E2 -21753.37} C_VEL
LIN {X 0,Y 216.288,Z 919.29,A -85,B 0,C 180,E1 -21755.013,E2 -21755.013} C_VEL
LIN {X 0,Y 210.337,Z 921.655,A -85,B 0,C 180,E1 -21758.436,E2 -21758.436} C_VEL
LIN {X 0,Y 207.657,Z 922.36,A -85,B 0,C 180,E1 -21760.218,E2 -21760.218} C_VEL
LIN {X 0,Y 202.935,Z 922.721,A -85,B 0,C 180,E1 -21763.916,E2 -21763.916} C_VEL
LIN {X 0,Y 199.034,Z 921.617,A -85,B 0,C 180,E1 -21767.768,E2 -21767.768} C_VEL
LIN {X 0,Y 197.589,Z 920.513,A -85,B 0,C 180,E1 -21769.756,E2 -21769.756} C_VEL
LIN {X 0,Y 195.246,Z 917.186,A -85,B 0,C 180,E1 -21773.801,E2 -21773.801} C_VEL
LIN {X 0,Y 193.983,Z 913.725,A -85,B 0,C 180,E1 -21776.885,E2 -21776.885} C_VEL
LIN {X 0,Y 192.931,Z 909.323,A -85,B 0,C 180,E1 -21780,E2 -21780} C_VEL
LIN {X 0,Y 192.582,Z 902.818,A -85,B 0,C 180,E1 -21783.662,E2 -21783.662} C_VEL
LIN {X 0,Y 192.753,Z 896.028,A -85,B 0,C 180,E1 -21786.806,E2 -21786.806} C_VEL
LIN {X 0,Y 193.419,Z 888.009,A -85,B 0,C 180,E1 -21789.939,E2 -21789.939} C_VEL
LIN {X 0,Y 194.262,Z 878.129,A -85,B 0,C 180,E1 -21793.068,E2 -21793.068} C_VEL
LIN {X 0,Y 195.422,Z 866.154,A -85,B 0,C 180,E1 -21796.184,E2 -21796.184} C_VEL
LIN {X 0,Y 196.659,Z 853.986,A -85,B 0,C 180,E1 -21798.762,E2 -21798.762} C_VEL
LIN {X 0,Y 197.141,Z 848.206,A -85,B 0,C 180,E1 -21799.796,E2 -21799.796} C_VEL
LIN {X 0,Y 194.529,Z 837.018,A -85,B 0,C 180,E1 -21801.65,E2 -21801.65} C_VEL
LIN {X 0,Y 192.691,Z 828.476,A -85,B 0,C 180,E1 -21802.943,E2 -21802.943} C_VEL
LIN {X 0,Y 192.603,Z 828.485,A -85,B 0,C 180,E1 -21808.86,E2 -21808.86} C_VEL
LIN {X 0,Y 192.603,Z 828.477,A -85,B 0,C 180,E1 -21813.185,E2 -21813.185} C_VEL
LIN {X 0,Y 192.55,Z 828.488,A -85,B 0,C 180,E1 -21818.353,E2 -21818.353} C_VEL
LIN {X 0,Y 192.492,Z 828.5,A -85,B 0,C 180,E1 -21823.091,E2 -21823.091} C_VEL
LIN {X 0,Y 192.491,Z 828.501,A -85,B 0,C 180,E1 -21826.905,E2 -21826.905} C_VEL
LIN {X 0,Y 192.574,Z 828.509,A -85,B 0,C 180,E1 -21830.976,E2 -21830.976} C_VEL
LIN {X 0,Y 193.541,Z 831.28,A -85,B 0,C 180,E1 -21831.53,E2 -21831.53} C_VEL
LIN {X 0,Y 198.012,Z 839.194,A -85,B 0,C 180,E1 -21833.619,E2 -21833.619} C_VEL
LIN {X 0,Y 201.959,Z 847.699,A -85,B 0,C 180,E1 -21835.829,E2 -21835.829} C_VEL
LIN {X 0,Y 205.455,Z 856.974,A -85,B 0,C 180,E1 -21838.299,E2 -21838.299} C_VEL
LIN {X 0,Y 207.893,Z 865.828,A -85,B 0,C 180,E1 -21840.754,E2 -21840.754} C_VEL
LIN {X 0,Y 209.028,Z 871.687,A -85,B 0,C 180,E1 -21842.482,E2 -21842.482} C_VEL
LIN {X 0,Y 208.684,Z 873.813,A -85,B 0,C 180,E1 -21842.996,E2 -21842.996} C_VEL
LIN {X 0,Y 206.133,Z 882.673,A -85,B 0,C 180,E1 -21845.31,E2 -21845.31} C_VEL
LIN {X 0,Y 203.056,Z 891.454,A -85,B 0,C 180,E1 -21848.153,E2 -21848.153} C_VEL
LIN {X 0,Y 200.811,Z 898.042,A -85,B 0,C 180,E1 -21850.901,E2 -21850.901} C_VEL
LIN {X 0,Y 199.002,Z 903.18,A -85,B 0,C 180,E1 -21853.585,E2 -21853.585} C_VEL
LIN {X 0,Y 196.917,Z 907.815,A -85,B 0,C 180,E1 -21856.582,E2 -21856.582} C_VEL
LIN {X 0,Y 195.392,Z 911.335,A -85,B 0,C 180,E1 -21859.636,E2 -21859.636} C_VEL
LIN {X 0,Y 194.776,Z 913.127,A -85,B 0,C 180,E1 -21861.698,E2 -21861.698} C_VEL
LIN {X 0,Y 194.326,Z 914.471,A -85,B 0,C 180,E1 -21863.768,E2 -21863.768} C_VEL
LIN {X 0,Y 193.573,Z 916.049,A -85,B 0,C 180,E1 -21867.916,E2 -21867.916} C_VEL
LIN {X 0,Y 193.473,Z 916.276,A -85,B 0,C 180,E1 -21869.996,E2 -21869.996} C_VEL
LIN {X 0,Y 193.874,Z 915.503,A -85,B 0,C 180,E1 -21874.154,E2 -21874.154} C_VEL
LIN {X 0,Y 194.292,Z 914.557,A -85,B 0,C 180,E1 -21876.226,E2 -21876.226} C_VEL
LIN {X 0,Y 194.705,Z 913.255,A -85,B 0,C 180,E1 -21878.298,E2 -21878.298} C_VEL
LIN {X 0,Y 195.816,Z 910.458,A -85,B 0,C 180,E1 -21881.381,E2 -21881.381} C_VEL
LIN {X 0,Y 197.629,Z 906.609,A -85,B 0,C 180,E1 -21884.41,E2 -21884.41} C_VEL
LIN {X 0,Y 199.589,Z 901.69,A -85,B 0,C 180,E1 -21887.412,E2 -21887.412} C_VEL
LIN {X 0,Y 201.785,Z 895.504,A -85,B 0,C 180,E1 -21890.379,E2 -21890.379} C_VEL
LIN {X 0,Y 204.492,Z 887.728,A -85,B 0,C 180,E1 -21893.276,E2 -21893.276} C_VEL
LIN {X 0,Y 207.033,Z 879.786,A -85,B 0,C 180,E1 -21895.642,E2 -21895.642} C_VEL
LIN {X 0,Y 209.264,Z 872.17,A -85,B 0,C 180,E1 -21897.498,E2 -21897.498} C_VEL
LIN {X 0,Y 207.153,Z 862.738,A -85,B 0,C 180,E1 -21900.266,E2 -21900.266} C_VEL
LIN {X 0,Y 204.449,Z 854.122,A -85,B 0,C 180,E1 -21902.628,E2 -21902.628} C_VEL
LIN {X 0,Y 201.066,Z 845.61,A -85,B 0,C 180,E1 -21904.87,E2 -21904.87} C_VEL
LIN {X 0,Y 196.545,Z 836.267,A -85,B 0,C 180,E1 -21907.288,E2 -21907.288} C_VEL
LIN {X 0,Y 194.847,Z 832.996,A -85,B 0,C 180,E1 -21908.119,E2 -21908.119} C_VEL
LIN {X 0,Y 193.019,Z 830.025,A -85,B 0,C 180,E1 -21908.921,E2 -21908.921} C_VEL
LIN {X 0,Y 192.653,Z 828.488,A -85,B 0,C 180,E1 -21909.255,E2 -21909.255} C_VEL
LIN {X 0,Y 192.619,Z 828.494,A -85,B 0,C 180,E1 -21913.881,E2 -21913.881} C_VEL
LIN {X 0,Y 192.605,Z 828.493,A -85,B 0,C 180,E1 -21918.943,E2 -21918.943} C_VEL
LIN {X 0,Y 192.616,Z 828.492,A -85,B 0,C 180,E1 -21923.383,E2 -21923.383} C_VEL
LIN {X 0,Y 192.596,Z 828.492,A -85,B 0,C 180,E1 -21927.057,E2 -21927.057} C_VEL
LIN {X 0,Y 192.653,Z 828.486,A -85,B 0,C 180,E1 -21931.69,E2 -21931.69} C_VEL
LIN {X 0,Y 192.693,Z 828.481,A -85,B 0,C 180,E1 -21936.347,E2 -21936.347} C_VEL
LIN {X 0,Y 192.719,Z 828.48,A -85,B 0,C 180,E1 -21941.456,E2 -21941.456} C_VEL
LIN {X 0,Y 192.758,Z 828.461,A -85,B 0,C 180,E1 -21945.213,E2 -21945.213} C_VEL
LIN {X 0,Y 192.967,Z 828.443,A -85,B 0,C 180,E1 -21949.508,E2 -21949.508} C_VEL
LIN {X 0,Y 193.047,Z 828.43,A -85,B 0,C 180,E1 -21951.627,E2 -21951.627} C_VEL
LIN {X 0,Y 193.248,Z 828.409,A -85,B 0,C 180,E1 -21957.916,E2 -21957.916} C_VEL
LIN {X 0,Y 193.428,Z 828.397,A -85,B 0,C 180,E1 -21960,E2 -21960} C_VEL
LIN {X 0,Y 192.958,Z 828.452,A -85,B 0,C 180,E1 -21964.177,E2 -21964.177} C_VEL
LIN {X 0,Y 193.045,Z 828.438,A -85,B 0,C 180,E1 -21968.373,E2 -21968.373} C_VEL
LIN {X 0,Y 192.796,Z 828.459,A -85,B 0,C 180,E1 -21972.634,E2 -21972.634} C_VEL
LIN {X 0,Y 192.743,Z 828.479,A -85,B 0,C 180,E1 -21976.96,E2 -21976.96} C_VEL
LIN {X 0,Y 192.606,Z 828.495,A -85,B 0,C 180,E1 -21981.401,E2 -21981.401} C_VEL
LIN {X 0,Y 192.63,Z 828.582,A -85,B 0,C 180,E1 -21985.095,E2 -21985.095} C_VEL
LIN {X 0,Y 193.522,Z 832.621,A -85,B 0,C 180,E1 -21989.365,E2 -21989.365} C_VEL
LIN {X 0,Y 194.549,Z 837.28,A -85,B 0,C 180,E1 -21993.82,E2 -21993.82} C_VEL
LIN {X 0,Y 195.387,Z 841.716,A -85,B 0,C 180,E1 -21997.697,E2 -21997.697} C_VEL
LIN {X 0,Y 196.195,Z 845.957,A -85,B 0,C 180,E1 -22001.221,E2 -22001.221} C_VEL
LIN {X 0,Y 197.226,Z 851.423,A -85,B 0,C 180,E1 -22005.454,E2 -22005.454} C_VEL
LIN {X 0,Y 198.065,Z 856.651,A -85,B 0,C 180,E1 -22009.306,E2 -22009.306} C_VEL
LIN {X 0,Y 197.56,Z 859.093,A -85,B 0,C 180,E1 -22010.968,E2 -22010.968} C_VEL
LIN {X 0,Y 200.537,Z 874.506,A -85,B 0,C 180,E1 -22012.737,E2 -22012.737} C_VEL
LIN {X 0,Y 202.132,Z 888.075,A -85,B 0,C 180,E1 -22014.541,E2 -22014.541} C_VEL
LIN {X 0,Y 202.611,Z 900.043,A -85,B 0,C 180,E1 -22016.356,E2 -22016.356} C_VEL
LIN {X 0,Y 202.293,Z 912.661,A -85,B 0,C 180,E1 -22018.597,E2 -22018.597} C_VEL
LIN {X 0,Y 201.367,Z 922.899,A -85,B 0,C 180,E1 -22020.755,E2 -22020.755} C_VEL
LIN {X 0,Y 200.129,Z 931.386,A -85,B 0,C 180,E1 -22022.841,E2 -22022.841} C_VEL
LIN {X 0,Y 198.486,Z 940.193,A -85,B 0,C 180,E1 -22025.419,E2 -22025.419} C_VEL
LIN {X 0,Y 196.913,Z 946.086,A -85,B 0,C 180,E1 -22027.443,E2 -22027.443} C_VEL
LIN {X 0,Y 194.921,Z 952.055,A -85,B 0,C 180,E1 -22029.851,E2 -22029.851} C_VEL
LIN {X 0,Y 193.138,Z 958.507,A -85,B 0,C 180,E1 -22033.08,E2 -22033.08} C_VEL
LIN {X 0,Y 192.055,Z 963.459,A -85,B 0,C 180,E1 -22036.244,E2 -22036.244} C_VEL
LIN {X 0,Y 191.525,Z 967.922,A -85,B 0,C 180,E1 -22040.061,E2 -22040.061} C_VEL
LIN {X 0,Y 190.898,Z 969.404,A -85,B 0,C 180,E1 -22041.767,E2 -22041.767} C_VEL
LIN {X 0,Y 189.44,Z 970.459,A -85,B 0,C 180,E1 -22043.476,E2 -22043.476} C_VEL
LIN {X 0,Y 186.183,Z 971.579,A -85,B 0,C 180,E1 -22046.989,E2 -22046.989} C_VEL
LIN {X 0,Y 185.454,Z 971.823,A -85,B 0,C 180,E1 -22048.821,E2 -22048.821} C_VEL
LIN {X 0,Y 185.482,Z 971.856,A -85,B 0,C 180,E1 -22049.437,E2 -22049.437} C_VEL
LIN {X 0,Y 185.594,Z 971.928,A -85,B 0,C 180,E1 -22050.004,E2 -22050.004} C_VEL
LIN {X 0,Y 185.274,Z 971.639,A -85,B 0,C 180,E1 -22052.178,E2 -22052.178} C_VEL
LIN {X 0,Y 184.996,Z 970.93,A -85,B 0,C 180,E1 -22054.361,E2 -22054.361} C_VEL
LIN {X 0,Y 184.534,Z 968.784,A -85,B 0,C 180,E1 -22058.022,E2 -22058.022} C_VEL
LIN {X 0,Y 184.789,Z 965.061,A -85,B 0,C 180,E1 -22062.078,E2 -22062.078} C_VEL
LIN {X 0,Y 185.13,Z 963.454,A -85,B 0,C 180,E1 -22063.449,E2 -22063.449} C_VEL
LIN {X 0,Y 186.473,Z 961.919,A -85,B 0,C 180,E1 -22067.552,E2 -22067.552} C_VEL
LIN {X 0,Y 189.163,Z 959.061,A -85,B 0,C 180,E1 -22071.814,E2 -22071.814} C_VEL
LIN {X 0,Y 192.206,Z 956.268,A -85,B 0,C 180,E1 -22074.87,E2 -22074.87} C_VEL
LIN {X 0,Y 197.257,Z 951.418,A -85,B 0,C 180,E1 -22078.754,E2 -22078.754} C_VEL
LIN {X 0,Y 202.75,Z 945.475,A -85,B 0,C 180,E1 -22082.502,E2 -22082.502} C_VEL
LIN {X 0,Y 209.383,Z 938.311,A -85,B 0,C 180,E1 -22085.976,E2 -22085.976} C_VEL
LIN {X 0,Y 215.03,Z 931.437,A -85,B 0,C 180,E1 -22088.992,E2 -22088.992} C_VEL
LIN {X 0,Y 222.094,Z 922.035,A -85,B 0,C 180,E1 -22092.919,E2 -22092.919} C_VEL
LIN {X 0,Y 228.24,Z 913.906,A -85,B 0,C 180,E1 -22096.357,E2 -22096.357} C_VEL
LIN {X 0,Y 230.866,Z 910.536,A -85,B 0,C 180,E1 -22097.954,E2 -22097.954} C_VEL
LIN {X 0,Y 231.938,Z 908.876,A -85,B 0,C 180,E1 -22099.251,E2 -22099.251} C_VEL
LIN {X 0,Y 232.522,Z 907.839,A -85,B 0,C 180,E1 -22100.6,E2 -22100.6} C_VEL
LIN {X 0,Y 232.772,Z 907.36,A -85,B 0,C 180,E1 -22101.725,E2 -22101.725} C_VEL
LIN {X 0,Y 232.692,Z 907.254,A -85,B 0,C 180,E1 -22102.839,E2 -22102.839} C_VEL
LIN {X 0,Y 231.653,Z 908.083,A -85,B 0,C 180,E1 -22105.003,E2 -22105.003} C_VEL
LIN {X 0,Y 230.583,Z 909.095,A -85,B 0,C 180,E1 -22105.964,E2 -22105.964} C_VEL
LIN {X 0,Y 222.941,Z 914.744,A -85,B 0,C 180,E1 -22108.658,E2 -22108.658} C_VEL
LIN {X 0,Y 215.977,Z 918.942,A -85,B 0,C 180,E1 -22111.479,E2 -22111.479} C_VEL
LIN {X 0,Y 210.204,Z 921.629,A -85,B 0,C 180,E1 -22114.237,E2 -22114.237} C_VEL
LIN {X 0,Y 207.044,Z 922.851,A -85,B 0,C 180,E1 -22115.963,E2 -22115.963} C_VEL
LIN {X 0,Y 201.216,Z 924.157,A -85,B 0,C 180,E1 -22119.557,E2 -22119.557} C_VEL
LIN {X 0,Y 196.269,Z 924.113,A -85,B 0,C 180,E1 -22123.354,E2 -22123.354} C_VEL
LIN {X 0,Y 192.194,Z 922.667,A -85,B 0,C 180,E1 -22127.326,E2 -22127.326} C_VEL
LIN {X 0,Y 189.254,Z 919.685,A -85,B 0,C 180,E1 -22131.458,E2 -22131.458} C_VEL
LIN {X 0,Y 187.313,Z 915.323,A -85,B 0,C 180,E1 -22135.697,E2 -22135.697} C_VEL
LIN {X 0,Y 186.138,Z 910.972,A -85,B 0,C 180,E1 -22138.918,E2 -22138.918} C_VEL
LIN {X 0,Y 185.621,Z 904.558,A -85,B 0,C 180,E1 -22142.713,E2 -22142.713} C_VEL
LIN {X 0,Y 185.543,Z 897.856,A -85,B 0,C 180,E1 -22145.979,E2 -22145.979} C_VEL
LIN {X 0,Y 186.215,Z 889.961,A -85,B 0,C 180,E1 -22149.23,E2 -22149.23} C_VEL
LIN {X 0,Y 186.733,Z 882.18,A -85,B 0,C 180,E1 -22151.873,E2 -22151.873} C_VEL
LIN {X 0,Y 187.486,Z 874.686,A -85,B 0,C 180,E1 -22154.103,E2 -22154.103} C_VEL
LIN {X 0,Y 188.441,Z 865.187,A -85,B 0,C 180,E1 -22156.522,E2 -22156.522} C_VEL
LIN {X 0,Y 189.444,Z 855.411,A -85,B 0,C 180,E1 -22158.661,E2 -22158.661} C_VEL
LIN {X 0,Y 190.036,Z 848.991,A -85,B 0,C 180,E1 -22159.855,E2 -22159.855} C_VEL
LIN {X 0,Y 187.288,Z 837.048,A -85,B 0,C 180,E1 -22161.881,E2 -22161.881} C_VEL
LIN {X 0,Y 185.659,Z 829.352,A -85,B 0,C 180,E1 -22163.052,E2 -22163.052} C_VEL
LIN {X 0,Y 185.526,Z 829.37,A -85,B 0,C 180,E1 -22169.503,E2 -22169.503} C_VEL
LIN {X 0,Y 185.537,Z 829.359,A -85,B 0,C 180,E1 -22173.551,E2 -22173.551} C_VEL
LIN {X 0,Y 185.508,Z 829.364,A -85,B 0,C 180,E1 -22177.313,E2 -22177.313} C_VEL
LIN {X 0,Y 185.469,Z 829.379,A -85,B 0,C 180,E1 -22180.719,E2 -22180.719} C_VEL
LIN {X 0,Y 185.462,Z 829.376,A -85,B 0,C 180,E1 -22186.055,E2 -22186.055} C_VEL
LIN {X 0,Y 185.466,Z 829.379,A -85,B 0,C 180,E1 -22189.116,E2 -22189.116} C_VEL
LIN {X 0,Y 186.358,Z 832.052,A -85,B 0,C 180,E1 -22189.681,E2 -22189.681} C_VEL
LIN {X 0,Y 187.829,Z 833.86,A -85,B 0,C 180,E1 -22190.309,E2 -22190.309} C_VEL
LIN {X 0,Y 193.165,Z 844.183,A -85,B 0,C 180,E1 -22193.172,E2 -22193.172} C_VEL
LIN {X 0,Y 197.003,Z 853.17,A -85,B 0,C 180,E1 -22195.689,E2 -22195.689} C_VEL
LIN {X 0,Y 199.949,Z 861.818,A -85,B 0,C 180,E1 -22198.178,E2 -22198.178} C_VEL
LIN {X 0,Y 202.121,Z 870.758,A -85,B 0,C 180,E1 -22200.866,E2 -22200.866} C_VEL
LIN {X 0,Y 202.626,Z 873.752,A -85,B 0,C 180,E1 -22201.816,E2 -22201.816} C_VEL
LIN {X 0,Y 200.352,Z 882.034,A -85,B 0,C 180,E1 -22203.99,E2 -22203.99} C_VEL
LIN {X 0,Y 197.525,Z 889.802,A -85,B 0,C 180,E1 -22206.401,E2 -22206.401} C_VEL
LIN {X 0,Y 194.753,Z 897.605,A -85,B 0,C 180,E1 -22209.538,E2 -22209.538} C_VEL
LIN {X 0,Y 192.276,Z 904.212,A -85,B 0,C 180,E1 -22212.994,E2 -22212.994} C_VEL
LIN {X 0,Y 190.092,Z 908.847,A -85,B 0,C 180,E1 -22216.091,E2 -22216.091} C_VEL
LIN {X 0,Y 188.486,Z 912.368,A -85,B 0,C 180,E1 -22219.252,E2 -22219.252} C_VEL
LIN {X 0,Y 187.833,Z 914.159,A -85,B 0,C 180,E1 -22221.389,E2 -22221.389} C_VEL
LIN {X 0,Y 187.348,Z 915.502,A -85,B 0,C 180,E1 -22223.535,E2 -22223.535} C_VEL
LIN {X 0,Y 186.554,Z 917.081,A -85,B 0,C 180,E1 -22227.837,E2 -22227.837} C_VEL
LIN {X 0,Y 186.449,Z 917.308,A -85,B 0,C 180,E1 -22229.996,E2 -22229.996} C_VEL
LIN {X 0,Y 186.869,Z 916.534,A -85,B 0,C 180,E1 -22234.31,E2 -22234.31} C_VEL
LIN {X 0,Y 187.313,Z 915.588,A -85,B 0,C 180,E1 -22236.459,E2 -22236.459} C_VEL
LIN {X 0,Y 187.771,Z 914.284,A -85,B 0,C 180,E1 -22238.606,E2 -22238.606} C_VEL
LIN {X 0,Y 188.934,Z 911.488,A -85,B 0,C 180,E1 -22241.801,E2 -22241.801} C_VEL
LIN {X 0,Y 190.833,Z 907.639,A -85,B 0,C 180,E1 -22244.935,E2 -22244.935} C_VEL
LIN {X 0,Y 192.897,Z 902.72,A -85,B 0,C 180,E1 -22248.036,E2 -22248.036} C_VEL
LIN {X 0,Y 195.214,Z 896.533,A -85,B 0,C 180,E1 -22251.097,E2 -22251.097} C_VEL
LIN {X 0,Y 198.062,Z 888.756,A -85,B 0,C 180,E1 -22254.079,E2 -22254.079} C_VEL
LIN {X 0,Y 200.724,Z 880.814,A -85,B 0,C 180,E1 -22256.51,E2 -22256.51} C_VEL
LIN {X 0,Y 202.772,Z 874.081,A -85,B 0,C 180,E1 -22258.221,E2 -22258.221} C_VEL
LIN {X 0,Y 201.051,Z 865.861,A -85,B 0,C 180,E1 -22260.784,E2 -22260.784} C_VEL
LIN {X 0,Y 198.698,Z 857.882,A -85,B 0,C 180,E1 -22263.137,E2 -22263.137} C_VEL
LIN {X 0,Y 195.049,Z 848.352,A -85,B 0,C 180,E1 -22265.832,E2 -22265.832} C_VEL
LIN {X 0,Y 191.553,Z 840.84,A -85,B 0,C 180,E1 -22267.924,E2 -22267.924} C_VEL
LIN {X 0,Y 187.429,Z 833.346,A -85,B 0,C 180,E1 -22270.044,E2 -22270.044} C_VEL
LIN {X 0,Y 185.872,Z 830.704,A -85,B 0,C 180,E1 -22270.805,E2 -22270.805} C_VEL
LIN {X 0,Y 185.575,Z 829.369,A -85,B 0,C 180,E1 -22271.064,E2 -22271.064} C_VEL
LIN {X 0,Y 185.577,Z 829.368,A -85,B 0,C 180,E1 -22276.011,E2 -22276.011} C_VEL
LIN {X 0,Y 185.573,Z 829.368,A -85,B 0,C 180,E1 -22279.922,E2 -22279.922} C_VEL
LIN {X 0,Y 185.565,Z 829.367,A -85,B 0,C 180,E1 -22282.701,E2 -22282.701} C_VEL
LIN {X 0,Y 185.534,Z 829.374,A -85,B 0,C 180,E1 -22287.973,E2 -22287.973} C_VEL
LIN {X 0,Y 185.57,Z 829.361,A -85,B 0,C 180,E1 -22290.573,E2 -22290.573} C_VEL
LIN {X 0,Y 185.575,Z 829.363,A -85,B 0,C 180,E1 -22295.38,E2 -22295.38} C_VEL
LIN {X 0,Y 185.662,Z 829.358,A -85,B 0,C 180,E1 -22301.132,E2 -22301.132} C_VEL
LIN {X 0,Y 185.75,Z 829.345,A -85,B 0,C 180,E1 -22306.878,E2 -22306.878} C_VEL
LIN {X 0,Y 185.994,Z 829.307,A -85,B 0,C 180,E1 -22311.307,E2 -22311.307} C_VEL
LIN {X 0,Y 186.193,Z 829.287,A -85,B 0,C 180,E1 -22317.837,E2 -22317.837} C_VEL
LIN {X 0,Y 186.392,Z 829.273,A -85,B 0,C 180,E1 -22320,E2 -22320} C_VEL
LIN {X 0,Y 185.905,Z 829.33,A -85,B 0,C 180,E1 -22324.336,E2 -22324.336} C_VEL
LIN {X 0,Y 185.993,Z 829.316,A -85,B 0,C 180,E1 -22328.693,E2 -22328.693} C_VEL
LIN {X 0,Y 185.72,Z 829.341,A -85,B 0,C 180,E1 -22333.123,E2 -22333.123} C_VEL
LIN {X 0,Y 185.676,Z 829.358,A -85,B 0,C 180,E1 -22337.626,E2 -22337.626} C_VEL
LIN {X 0,Y 185.64,Z 829.536,A -85,B 0,C 180,E1 -22343.718,E2 -22343.718} C_VEL
LIN {X 0,Y 186.443,Z 833.477,A -85,B 0,C 180,E1 -22348.111,E2 -22348.111} C_VEL
LIN {X 0,Y 187.474,Z 838.205,A -85,B 0,C 180,E1 -22352.927,E2 -22352.927} C_VEL
LIN {X 0,Y 188.471,Z 843.309,A -85,B 0,C 180,E1 -22357.602,E2 -22357.602} C_VEL
LIN {X 0,Y 189.477,Z 848.614,A -85,B 0,C 180,E1 -22362.119,E2 -22362.119} C_VEL
LIN {X 0,Y 190.46,Z 853.897,A -85,B 0,C 180,E1 -22366.326,E2 -22366.326} C_VEL
LIN {X 0,Y 191.011,Z 857.885,A -85,B 0,C 180,E1 -22369.354,E2 -22369.354} C_VEL
LIN {X 0,Y 191.906,Z 861.7,A -85,B 0,C 180,E1 -22369.829,E2 -22369.829} C_VEL
LIN {X 0,Y 194.251,Z 873.821,A -85,B 0,C 180,E1 -22371.361,E2 -22371.361} C_VEL
LIN {X 0,Y 195.803,Z 887.126,A -85,B 0,C 180,E1 -22373.237,E2 -22373.237} C_VEL
LIN {X 0,Y 196.245,Z 898.536,A -85,B 0,C 180,E1 -22375.046,E2 -22375.046} C_VEL
LIN {X 0,Y 195.909,Z 910.507,A -85,B 0,C 180,E1 -22377.235,E2 -22377.235} C_VEL
LIN {X 0,Y 195.03,Z 920.626,A -85,B 0,C 180,E1 -22379.407,E2 -22379.407} C_VEL
LIN {X 0,Y 193.592,Z 930.306,A -85,B 0,C 180,E1 -22381.844,E2 -22381.844} C_VEL
LIN {X 0,Y 191.842,Z 939.119,A -85,B 0,C 180,E1 -22384.508,E2 -22384.508} C_VEL
LIN {X 0,Y 190.806,Z 943.648,A -85,B 0,C 180,E1 -22386.103,E2 -22386.103} C_VEL
LIN {X 0,Y 188.087,Z 951.475,A -85,B 0,C 180,E1 -22389.316,E2 -22389.316} C_VEL
LIN {X 0,Y 186.264,Z 957.452,A -85,B 0,C 180,E1 -22392.436,E2 -22392.436} C_VEL
LIN {X 0,Y 185.086,Z 962.405,A -85,B 0,C 180,E1 -22395.715,E2 -22395.715} C_VEL
LIN {X 0,Y 184.526,Z 966.254,A -85,B 0,C 180,E1 -22399.026,E2 -22399.026} C_VEL
LIN {X 0,Y 184.531,Z 968.826,A -85,B 0,C 180,E1 -22401.984,E2 -22401.984} C_VEL
LIN {X 0,Y 184.975,Z 970.951,A -85,B 0,C 180,E1 -22405.646,E2 -22405.646} C_VEL
LIN {X 0,Y 185.266,Z 971.652,A -85,B 0,C 180,E1 -22407.83,E2 -22407.83} C_VEL
LIN {X 0,Y 185.482,Z 971.856,A -85,B 0,C 180,E1 -22409.437,E2 -22409.437} C_VEL
LIN {X 0,Y 185.283,Z 971.864,A -85,B 0,C 180,E1 -22410.641,E2 -22410.641} C_VEL
LIN {X 0,Y 183.845,Z 971.429,A -85,B 0,C 180,E1 -22412.412,E2 -22412.412} C_VEL
LIN {X 0,Y 180.172,Z 969.885,A -85,B 0,C 180,E1 -22415.314,E2 -22415.314} C_VEL
LIN {X 0,Y 177.834,Z 968.196,A -85,B 0,C 180,E1 -22417.744,E2 -22417.744} C_VEL
LIN {X 0,Y 177.458,Z 967.26,A -85,B 0,C 180,E1 -22419.007,E2 -22419.007} C_VEL
LIN {X 0,Y 177.817,Z 964.013,A -85,B 0,C 180,E1 -22422.559,E2 -22422.559} C_VEL
LIN {X 0,Y 178.36,Z 961.925,A -85,B 0,C 180,E1 -22424.552,E2 -22424.552} C_VEL
LIN {X 0,Y 179.693,Z 960.797,A -85,B 0,C 180,E1 -22428.237,E2 -22428.237} C_VEL
LIN {X 0,Y 182.584,Z 958.343,A -85,B 0,C 180,E1 -22432.643,E2 -22432.643} C_VEL
LIN {X 0,Y 188.301,Z 953.631,A -85,B 0,C 180,E1 -22437.814,E2 -22437.814} C_VEL
LIN {X 0,Y 192.359,Z 950.064,A -85,B 0,C 180,E1 -22440.768,E2 -22440.768} C_VEL
LIN {X 0,Y 200.127,Z 942.671,A -85,B 0,C 180,E1 -22445.415,E2 -22445.415} C_VEL
LIN {X 0,Y 206.245,Z 936.602,A -85,B 0,C 180,E1 -22448.395,E2 -22448.395} C_VEL
LIN {X 0,Y 213.769,Z 928.015,A -85,B 0,C 180,E1 -22452.378,E2 -22452.378} C_VEL
LIN {X 0,Y 220.372,Z 920.351,A -85,B 0,C 180,E1 -22455.856,E2 -22455.856} C_VEL
LIN {X 0,Y 225.26,Z 914.681,A -85,B 0,C 180,E1 -22458.489,E2 -22458.489} C_VEL
LIN {X 0,Y 226.056,Z 913.64,A -85,B 0,C 180,E1 -22459.241,E2 -22459.241} C_VEL
LIN {X 0,Y 226.951,Z 912.286,A -85,B 0,C 180,E1 -22460.734,E2 -22460.734} C_VEL
LIN {X 0,Y 227.211,Z 911.771,A -85,B 0,C 180,E1 -22461.784,E2 -22461.784} C_VEL
LIN {X 0,Y 226.512,Z 912.059,A -85,B 0,C 180,E1 -22463.877,E2 -22463.877} C_VEL
LIN {X 0,Y 225.93,Z 912.417,A -85,B 0,C 180,E1 -22464.735,E2 -22464.735} C_VEL
LIN {X 0,Y 221.63,Z 915.311,A -85,B 0,C 180,E1 -22466.294,E2 -22466.294} C_VEL
LIN {X 0,Y 213.661,Z 919.999,A -85,B 0,C 180,E1 -22469.206,E2 -22469.206} C_VEL
LIN {X 0,Y 207.73,Z 922.736,A -85,B 0,C 180,E1 -22471.728,E2 -22471.728} C_VEL
LIN {X 0,Y 200.866,Z 924.918,A -85,B 0,C 180,E1 -22475.174,E2 -22475.174} C_VEL
LIN {X 0,Y 197.72,Z 925.565,A -85,B 0,C 180,E1 -22476.983,E2 -22476.983} C_VEL
LIN {X 0,Y 192.078,Z 925.84,A -85,B 0,C 180,E1 -22480.773,E2 -22480.773} C_VEL
LIN {X 0,Y 187.361,Z 924.681,A -85,B 0,C 180,E1 -22484.777,E2 -22484.777} C_VEL
LIN {X 0,Y 185.348,Z 923.588,A -85,B 0,C 180,E1 -22486.85,E2 -22486.85} C_VEL
LIN {X 0,Y 182.29,Z 920.302,A -85,B 0,C 180,E1 -22491.129,E2 -22491.129} C_VEL
LIN {X 0,Y 180.246,Z 915.453,A -85,B 0,C 180,E1 -22495.528,E2 -22495.528} C_VEL
LIN {X 0,Y 179.041,Z 910.818,A -85,B 0,C 180,E1 -22498.876,E2 -22498.876} C_VEL
LIN {X 0,Y 178.593,Z 905.167,A -85,B 0,C 180,E1 -22502.255,E2 -22502.255} C_VEL
LIN {X 0,Y 178.448,Z 898.357,A -85,B 0,C 180,E1 -22505.651,E2 -22505.651} C_VEL
LIN {X 0,Y 179.083,Z 890.105,A -85,B 0,C 180,E1 -22509.129,E2 -22509.129} C_VEL
LIN {X 0,Y 180.063,Z 878.157,A -85,B 0,C 180,E1 -22513.164,E2 -22513.164} C_VEL
LIN {X 0,Y 181.144,Z 867.572,A -85,B 0,C 180,E1 -22516.048,E2 -22516.048} C_VEL
LIN {X 0,Y 182.228,Z 856.698,A -85,B 0,C 180,E1 -22518.553,E2 -22518.553} C_VEL
LIN {X 0,Y 182.894,Z 849.498,A -85,B 0,C 180,E1 -22519.94,E2 -22519.94} C_VEL
LIN {X 0,Y 180.417,Z 838.823,A -85,B 0,C 180,E1 -22521.827,E2 -22521.827} C_VEL
LIN {X 0,Y 178.613,Z 830.23,A -85,B 0,C 180,E1 -22523.171,E2 -22523.171} C_VEL
LIN {X 0,Y 178.473,Z 830.251,A -85,B 0,C 180,E1 -22529.959,E2 -22529.959} C_VEL
LIN {X 0,Y 178.491,Z 830.241,A -85,B 0,C 180,E1 -22534.216,E2 -22534.216} C_VEL
LIN {X 0,Y 178.396,Z 830.255,A -85,B 0,C 180,E1 -22539.075,E2 -22539.075} C_VEL
LIN {X 0,Y 178.401,Z 830.252,A -85,B 0,C 180,E1 -22542.045,E2 -22542.045} C_VEL
LIN {X 0,Y 178.424,Z 830.317,A -85,B 0,C 180,E1 -22547.083,E2 -22547.083} C_VEL
LIN {X 0,Y 179.343,Z 832.999,A -85,B 0,C 180,E1 -22547.694,E2 -22547.694} C_VEL
LIN {X 0,Y 180.871,Z 834.924,A -85,B 0,C 180,E1 -22548.417,E2 -22548.417} C_VEL
LIN {X 0,Y 186.702,Z 845.877,A -85,B 0,C 180,E1 -22551.754,E2 -22551.754} C_VEL
LIN {X 0,Y 190.377,Z 854.32,A -85,B 0,C 180,E1 -22554.308,E2 -22554.308} C_VEL
LIN {X 0,Y 193.337,Z 862.974,A -85,B 0,C 180,E1 -22556.953,E2 -22556.953} C_VEL
LIN {X 0,Y 195.542,Z 871.873,A -85,B 0,C 180,E1 -22559.786,E2 -22559.786} C_VEL
LIN {X 0,Y 196.138,Z 875.387,A -85,B 0,C 180,E1 -22560.956,E2 -22560.956} C_VEL
LIN {X 0,Y 196.061,Z 876.541,A -85,B 0,C 180,E1 -22561.299,E2 -22561.299} C_VEL
LIN {X 0,Y 192.881,Z 886.335,A -85,B 0,C 180,E1 -22564.068,E2 -22564.068} C_VEL
LIN {X 0,Y 190.089,Z 893.521,A -85,B 0,C 180,E1 -22566.577,E2 -22566.577} C_VEL
LIN {X 0,Y 187.713,Z 899.878,A -85,B 0,C 180,E1 -22569.392,E2 -22569.392} C_VEL
LIN {X 0,Y 185.573,Z 905.244,A -85,B 0,C 180,E1 -22572.36,E2 -22572.36} C_VEL
LIN {X 0,Y 183.282,Z 909.879,A -85,B 0,C 180,E1 -22575.563,E2 -22575.563} C_VEL
LIN {X 0,Y 181.588,Z 913.4,A -85,B 0,C 180,E1 -22578.838,E2 -22578.838} C_VEL
LIN {X 0,Y 180.895,Z 915.19,A -85,B 0,C 180,E1 -22581.056,E2 -22581.056} C_VEL
LIN {X 0,Y 180.372,Z 916.533,A -85,B 0,C 180,E1 -22583.283,E2 -22583.283} C_VEL
LIN {X 0,Y 179.535,Z 918.112,A -85,B 0,C 180,E1 -22587.753,E2 -22587.753} C_VEL
LIN {X 0,Y 179.425,Z 918.339,A -85,B 0,C 180,E1 -22589.996,E2 -22589.996} C_VEL
LIN {X 0,Y 179.865,Z 917.565,A -85,B 0,C 180,E1 -22594.478,E2 -22594.478} C_VEL
LIN {X 0,Y 180.339,Z 916.618,A -85,B 0,C 180,E1 -22596.71,E2 -22596.71} C_VEL
LIN {X 0,Y 180.841,Z 915.312,A -85,B 0,C 180,E1 -22598.939,E2 -22598.939} C_VEL
LIN {X 0,Y 182.063,Z 912.519,A -85,B 0,C 180,E1 -22602.254,E2 -22602.254} C_VEL
LIN {X 0,Y 184.054,Z 908.67,A -85,B 0,C 180,E1 -22605.499,E2 -22605.499} C_VEL
LIN {X 0,Y 186.235,Z 903.749,A -85,B 0,C 180,E1 -22608.705,E2 -22608.705} C_VEL
LIN {X 0,Y 188.699,Z 897.559,A -85,B 0,C 180,E1 -22611.862,E2 -22611.862} C_VEL
LIN {X 0,Y 191.067,Z 891.243,A -85,B 0,C 180,E1 -22614.44,E2 -22614.44} C_VEL
LIN {X 0,Y 193.92,Z 883.58,A -85,B 0,C 180,E1 -22616.933,E2 -22616.933} C_VEL
LIN {X 0,Y 196.292,Z 875.729,A -85,B 0,C 180,E1 -22619.073,E2 -22619.073} C_VEL
LIN {X 0,Y 194.445,Z 866.833,A -85,B 0,C 180,E1 -22621.991,E2 -22621.991} C_VEL
LIN {X 0,Y 192.057,Z 858.953,A -85,B 0,C 180,E1 -22624.461,E2 -22624.461} C_VEL
LIN {X 0,Y 188.963,Z 850.926,A -85,B 0,C 180,E1 -22626.902,E2 -22626.902} C_VEL
LIN {X 0,Y 184.897,Z 842.129,A -85,B 0,C 180,E1 -22629.541,E2 -22629.541} C_VEL
LIN {X 0,Y 180.59,Z 834.461,A -85,B 0,C 180,E1 -22631.919,E2 -22631.919} C_VEL
LIN {X 0,Y 178.964,Z 831.984,A -85,B 0,C 180,E1 -22632.751,E2 -22632.751} C_VEL
LIN {X 0,Y 178.544,Z 830.245,A -85,B 0,C 180,E1 -22633.132,E2 -22633.132} C_VEL
LIN {X 0,Y 178.513,Z 830.244,A -85,B 0,C 180,E1 -22638.412,E2 -22638.412} C_VEL
LIN {X 0,Y 178.478,Z 830.253,A -85,B 0,C 180,E1 -22643.796,E2 -22643.796} C_VEL
LIN {X 0,Y 178.48,Z 830.246,A -85,B 0,C 180,E1 -22646.545,E2 -22646.545} C_VEL
LIN {X 0,Y 178.511,Z 830.239,A -85,B 0,C 180,E1 -22650.004,E2 -22650.004} C_VEL
LIN {X 0,Y 178.512,Z 830.24,A -85,B 0,C 180,E1 -22654.88,E2 -22654.88} C_VEL
LIN {X 0,Y 178.61,Z 830.233,A -85,B 0,C 180,E1 -22660.782,E2 -22660.782} C_VEL
LIN {X 0,Y 178.667,Z 830.223,A -85,B 0,C 180,E1 -22666.348,E2 -22666.348} C_VEL
LIN {X 0,Y 178.923,Z 830.187,A -85,B 0,C 180,E1 -22670.96,E2 -22670.96} C_VEL
LIN {X 0,Y 179.138,Z 830.165,A -85,B 0,C 180,E1 -22677.751,E2 -22677.751} C_VEL
LIN {X 0,Y 179.355,Z 830.15,A -85,B 0,C 180,E1 -22680,E2 -22680} C_VEL
LIN {X 0,Y 178.854,Z 830.209,A -85,B 0,C 180,E1 -22684.507,E2 -22684.507} C_VEL
LIN {X 0,Y 178.922,Z 830.196,A -85,B 0,C 180,E1 -22689.04,E2 -22689.04} C_VEL
LIN {X 0,Y 178.647,Z 830.226,A -85,B 0,C 180,E1 -22693.653,E2 -22693.653} C_VEL
LIN {X 0,Y 178.608,Z 830.24,A -85,B 0,C 180,E1 -22699.216,E2 -22699.216} C_VEL
LIN {X 0,Y 178.531,Z 830.305,A -85,B 0,C 180,E1 -22701.961,E2 -22701.961} C_VEL
LIN {X 0,Y 179.422,Z 834.324,A -85,B 0,C 180,E1 -22706.773,E2 -22706.773} C_VEL
LIN {X 0,Y 180.419,Z 838.957,A -85,B 0,C 180,E1 -22711.745,E2 -22711.745} C_VEL
LIN {X 0,Y 181.468,Z 844.234,A -85,B 0,C 180,E1 -22716.891,E2 -22716.891} C_VEL
LIN {X 0,Y 182.514,Z 850.013,A -85,B 0,C 180,E1 -22722.003,E2 -22722.003} C_VEL
LIN {X 0,Y 183.577,Z 855.626,A -85,B 0,C 180,E1 -22726.668,E2 -22726.668} C_VEL
LIN {X 0,Y 183.757,Z 856.553,A -85,B 0,C 180,E1 -22727.412,E2 -22727.412} C_VEL
LIN {X 0,Y 185.032,Z 860.34,A -85,B 0,C 180,E1 -22728.004,E2 -22728.004} C_VEL
LIN {X 0,Y 185.953,Z 862.445,A -85,B 0,C 180,E1 -22728.407,E2 -22728.407} C_VEL
LIN {X 0,Y 187.994,Z 872.283,A -85,B 0,C 180,E1 -22729.781,E2 -22729.781} C_VEL
LIN {X 0,Y 189.516,Z 885.853,A -85,B 0,C 180,E1 -22731.787,E2 -22731.787} C_VEL
LIN {X 0,Y 189.994,Z 897.414,A -85,B 0,C 180,E1 -22733.717,E2 -22733.717} C_VEL
LIN {X 0,Y 189.628,Z 908.713,A -85,B 0,C 180,E1 -22735.858,E2 -22735.858} C_VEL
LIN {X 0,Y 188.658,Z 919.536,A -85,B 0,C 180,E1 -22738.256,E2 -22738.256} C_VEL
LIN {X 0,Y 187.147,Z 929.23,A -85,B 0,C 180,E1 -22740.783,E2 -22740.783} C_VEL
LIN {X 0,Y 185.284,Z 938.05,A -85,B 0,C 180,E1 -22743.537,E2 -22743.537} C_VEL
LIN {X 0,Y 183.793,Z 943.992,A -85,B 0,C 180,E1 -22745.733,E2 -22745.733} C_VEL
LIN {X 0,Y 181.27,Z 950.896,A -85,B 0,C 180,E1 -22748.741,E2 -22748.741} C_VEL
LIN {X 0,Y 179.409,Z 956.395,A -85,B 0,C 180,E1 -22751.741,E2 -22751.741} C_VEL
LIN {X 0,Y 178.147,Z 961.354,A -85,B 0,C 180,E1 -22755.146,E2 -22755.146} C_VEL
LIN {X 0,Y 177.506,Z 965.204,A -85,B 0,C 180,E1 -22758.586,E2 -22758.586} C_VEL
LIN {X 0,Y 177.489,Z 967.918,A -85,B 0,C 180,E1 -22761.859,E2 -22761.859} C_VEL
LIN {X 0,Y 177.876,Z 969.906,A -85,B 0,C 180,E1 -22765.472,E2 -22765.472} C_VEL
LIN {X 0,Y 178.204,Z 970.614,A -85,B 0,C 180,E1 -22767.744,E2 -22767.744} C_VEL
LIN {X 0,Y 178.552,Z 970.894,A -85,B 0,C 180,E1 -22770.004,E2 -22770.004} C_VEL
LIN {X 0,Y 178.213,Z 970.602,A -85,B 0,C 180,E1 -22772.264,E2 -22772.264} C_VEL
LIN {X 0,Y 177.896,Z 969.884,A -85,B 0,C 180,E1 -22774.536,E2 -22774.536} C_VEL
LIN {X 0,Y 177.458,Z 967.26,A -85,B 0,C 180,E1 -22779.007,E2 -22779.007} C_VEL
LIN {X 0,Y 176.788,Z 966.235,A -85,B 0,C 180,E1 -22780.236,E2 -22780.236} C_VEL
LIN {X 0,Y 171.689,Z 961.89,A -85,B 0,C 180,E1 -22784.094,E2 -22784.094} C_VEL
LIN {X 0,Y 171.598,Z 960.422,A -85,B 0,C 180,E1 -22785.348,E2 -22785.348} C_VEL
LIN {X 0,Y 172.95,Z 959.539,A -85,B 0,C 180,E1 -22788.975,E2 -22788.975} C_VEL
LIN {X 0,Y 176.058,Z 957.427,A -85,B 0,C 180,E1 -22793.531,E2 -22793.531} C_VEL
LIN {X 0,Y 180.695,Z 954.176,A -85,B 0,C 180,E1 -22797.826,E2 -22797.826} C_VEL
LIN {X 0,Y 186.235,Z 949.891,A -85,B 0,C 180,E1 -22801.896,E2 -22801.896} C_VEL
LIN {X 0,Y 194.403,Z 943.166,A -85,B 0,C 180,E1 -22806.624,E2 -22806.624} C_VEL
LIN {X 0,Y 200.671,Z 937.682,A -85,B 0,C 180,E1 -22809.602,E2 -22809.602} C_VEL
LIN {X 0,Y 208.682,Z 929.596,A -85,B 0,C 180,E1 -22813.666,E2 -22813.666} C_VEL
LIN {X 0,Y 215.627,Z 922.421,A -85,B 0,C 180,E1 -22817.17,E2 -22817.17} C_VEL
LIN {X 0,Y 219.117,Z 918.969,A -85,B 0,C 180,E1 -22818.903,E2 -22818.903} C_VEL
LIN {X 0,Y 220.565,Z 917.458,A -85,B 0,C 180,E1 -22819.887,E2 -22819.887} C_VEL
LIN {X 0,Y 220.938,Z 916.916,A -85,B 0,C 180,E1 -22820.491,E2 -22820.491} C_VEL
LIN {X 0,Y 221.038,Z 916.024,A -85,B 0,C 180,E1 -22822.835,E2 -22822.835} C_VEL
LIN {X 0,Y 220.81,Z 916.035,A -85,B 0,C 180,E1 -22823.495,E2 -22823.495} C_VEL
LIN {X 0,Y 218.546,Z 917.409,A -85,B 0,C 180,E1 -22824.631,E2 -22824.631} C_VEL
LIN {X 0,Y 209.819,Z 922.033,A -85,B 0,C 180,E1 -22827.593,E2 -22827.593} C_VEL
LIN {X 0,Y 205.735,Z 923.786,A -85,B 0,C 180,E1 -22829.176,E2 -22829.176} C_VEL
LIN {X 0,Y 198.176,Z 926.278,A -85,B 0,C 180,E1 -22832.547,E2 -22832.547} C_VEL
LIN {X 0,Y 191.414,Z 927.388,A -85,B 0,C 180,E1 -22836.179,E2 -22836.179} C_VEL
LIN {X 0,Y 185.52,Z 927.241,A -85,B 0,C 180,E1 -22840.066,E2 -22840.066} C_VEL
LIN {X 0,Y 180.595,Z 925.721,A -85,B 0,C 180,E1 -22844.192,E2 -22844.192} C_VEL
LIN {X 0,Y 178.492,Z 924.397,A -85,B 0,C 180,E1 -22846.335,E2 -22846.335} C_VEL
LIN {X 0,Y 175.289,Z 920.678,A -85,B 0,C 180,E1 -22850.771,E2 -22850.771} C_VEL
LIN {X 0,Y 173.626,Z 916.974,A -85,B 0,C 180,E1 -22854.192,E2 -22854.192} C_VEL
LIN {X 0,Y 172.294,Z 912.371,A -85,B 0,C 180,E1 -22857.662,E2 -22857.662} C_VEL
LIN {X 0,Y 171.581,Z 906.767,A -85,B 0,C 180,E1 -22861.174,E2 -22861.174} C_VEL
LIN {X 0,Y 171.358,Z 900.038,A -85,B 0,C 180,E1 -22864.705,E2 -22864.705} C_VEL
LIN {X 0,Y 171.744,Z 892.136,A -85,B 0,C 180,E1 -22868.235,E2 -22868.235} C_VEL
LIN {X 0,Y 172.336,Z 884.161,A -85,B 0,C 180,E1 -22871.166,E2 -22871.166} C_VEL
LIN {X 0,Y 173.271,Z 874.961,A -85,B 0,C 180,E1 -22874.085,E2 -22874.085} C_VEL
LIN {X 0,Y 174.247,Z 865.219,A -85,B 0,C 180,E1 -22876.701,E2 -22876.701} C_VEL
LIN {X 0,Y 175.465,Z 853.709,A -85,B 0,C 180,E1 -22879.296,E2 -22879.296} C_VEL
LIN {X 0,Y 175.783,Z 850.732,A -85,B 0,C 180,E1 -22879.867,E2 -22879.867} C_VEL
LIN {X 0,Y 173.357,Z 839.755,A -85,B 0,C 180,E1 -22881.875,E2 -22881.875} C_VEL
LIN {X 0,Y 171.563,Z 831.109,A -85,B 0,C 180,E1 -22883.3,E2 -22883.3} C_VEL
LIN {X 0,Y 171.401,Z 831.129,A -85,B 0,C 180,E1 -22889.475,E2 -22889.475} C_VEL
LIN {X 0,Y 171.401,Z 831.131,A -85,B 0,C 180,E1 -22895.033,E2 -22895.033} C_VEL
LIN {X 0,Y 171.351,Z 831.13,A -85,B 0,C 180,E1 -22898.799,E2 -22898.799} C_VEL
LIN {X 0,Y 171.343,Z 831.142,A -85,B 0,C 180,E1 -22904.555,E2 -22904.555} C_VEL
LIN {X 0,Y 171.384,Z 831.321,A -85,B 0,C 180,E1 -22904.801,E2 -22904.801} C_VEL
LIN {X 0,Y 172.377,Z 834.009,A -85,B 0,C 180,E1 -22905.492,E2 -22905.492} C_VEL
LIN {X 0,Y 174.126,Z 836.32,A -85,B 0,C 180,E1 -22906.421,E2 -22906.421} C_VEL
LIN {X 0,Y 179.436,Z 845.908,A -85,B 0,C 180,E1 -22909.664,E2 -22909.664} C_VEL
LIN {X 0,Y 183.523,Z 854.927,A -85,B 0,C 180,E1 -22912.621,E2 -22912.621} C_VEL
LIN {X 0,Y 186.747,Z 864.142,A -85,B 0,C 180,E1 -22915.628,E2 -22915.628} C_VEL
LIN {X 0,Y 188.785,Z 871.951,A -85,B 0,C 180,E1 -22918.271,E2 -22918.271} C_VEL
LIN {X 0,Y 189.788,Z 877.932,A -85,B 0,C 180,E1 -22920.37,E2 -22920.37} C_VEL
LIN {X 0,Y 186.59,Z 887.368,A -85,B 0,C 180,E1 -22923.125,E2 -22923.125} C_VEL
LIN {X 0,Y 183.664,Z 894.555,A -85,B 0,C 180,E1 -22925.706,E2 -22925.706} C_VEL
LIN {X 0,Y 181.21,Z 900.81,A -85,B 0,C 180,E1 -22928.562,E2 -22928.562} C_VEL
LIN {X 0,Y 178.894,Z 906.277,A -85,B 0,C 180,E1 -22931.678,E2 -22931.678} C_VEL
LIN {X 0,Y 176.489,Z 910.912,A -85,B 0,C 180,E1 -22934.995,E2 -22934.995} C_VEL
LIN {X 0,Y 174.702,Z 914.432,A -85,B 0,C 180,E1 -22938.392,E2 -22938.392} C_VEL
LIN {X 0,Y 173.963,Z 916.221,A -85,B 0,C 180,E1 -22940.696,E2 -22940.696} C_VEL
LIN {X 0,Y 173.4,Z 917.565,A -85,B 0,C 180,E1 -22943.012,E2 -22943.012} C_VEL
LIN {X 0,Y 172.517,Z 919.143,A -85,B 0,C 180,E1 -22947.661,E2 -22947.661} C_VEL
LIN {X 0,Y 172.402,Z 919.37,A -85,B 0,C 180,E1 -22949.996,E2 -22949.996} C_VEL
LIN {X 0,Y 172.863,Z 918.596,A -85,B 0,C 180,E1 -22954.66,E2 -22954.66} C_VEL
LIN {X 0,Y 173.368,Z 917.648,A -85,B 0,C 180,E1 -22956.981,E2 -22956.981} C_VEL
LIN {X 0,Y 173.915,Z 916.342,A -85,B 0,C 180,E1 -22959.298,E2 -22959.298} C_VEL
LIN {X 0,Y 175.205,Z 913.549,A -85,B 0,C 180,E1 -22962.741,E2 -22962.741} C_VEL
LIN {X 0,Y 177.294,Z 909.7,A -85,B 0,C 180,E1 -22966.106,E2 -22966.106} C_VEL
LIN {X 0,Y 179.602,Z 904.778,A -85,B 0,C 180,E1 -22969.423,E2 -22969.423} C_VEL
LIN {X 0,Y 182.202,Z 898.587,A -85,B 0,C 180,E1 -22972.684,E2 -22972.684} C_VEL
LIN {X 0,Y 184.695,Z 892.272,A -85,B 0,C 180,E1 -22975.341,E2 -22975.341} C_VEL
LIN {X 0,Y 187.685,Z 884.609,A -85,B 0,C 180,E1 -22977.904,E2 -22977.904} C_VEL
LIN {X 0,Y 189.798,Z 878.338,A -85,B 0,C 180,E1 -22979.66,E2 -22979.66} C_VEL
LIN {X 0,Y 188.703,Z 871.502,A -85,B 0,C 180,E1 -22982.049,E2 -22982.049} C_VEL
LIN {X 0,Y 186.654,Z 863.79,A -85,B 0,C 180,E1 -22984.659,E2 -22984.659} C_VEL
LIN {X 0,Y 183.677,Z 855.298,A -85,B 0,C 180,E1 -22987.443,E2 -22987.443} C_VEL
LIN {X 0,Y 180.147,Z 847.219,A -85,B 0,C 180,E1 -22990.08,E2 -22990.08} C_VEL
LIN {X 0,Y 175.412,Z 838.624,A -85,B 0,C 180,E1 -22993.013,E2 -22993.013} C_VEL
LIN {X 0,Y 173.733,Z 835.481,A -85,B 0,C 180,E1 -22994.03,E2 -22994.03} C_VEL
LIN {X 0,Y 172.076,Z 833.204,A -85,B 0,C 180,E1 -22994.932,E2 -22994.932} C_VEL
LIN {X 0,Y 171.476,Z 831.126,A -85,B 0,C 180,E1 -22995.467,E2 -22995.467} C_VEL
LIN {X 0,Y 171.436,Z 831.121,A -85,B 0,C 180,E1 -23001.152,E2 -23001.152} C_VEL
LIN {X 0,Y 171.43,Z 831.122,A -85,B 0,C 180,E1 -23005.069,E2 -23005.069} C_VEL
LIN {X 0,Y 171.437,Z 831.121,A -85,B 0,C 180,E1 -23010.532,E2 -23010.532} C_VEL
LIN {X 0,Y 171.44,Z 831.126,A -85,B 0,C 180,E1 -23015.799,E2 -23015.799} C_VEL
LIN {X 0,Y 171.566,Z 831.111,A -85,B 0,C 180,E1 -23020.87,E2 -23020.87} C_VEL
LIN {X 0,Y 171.58,Z 831.101,A -85,B 0,C 180,E1 -23025.773,E2 -23025.773} C_VEL
LIN {X 0,Y 171.859,Z 831.067,A -85,B 0,C 180,E1 -23030.585,E2 -23030.585} C_VEL
LIN {X 0,Y 171.806,Z 831.083,A -85,B 0,C 180,E1 -23035.307,E2 -23035.307} C_VEL
LIN {X 0,Y 172.318,Z 831.027,A -85,B 0,C 180,E1 -23040,E2 -23040} C_VEL
LIN {X 0,Y 171.803,Z 831.088,A -85,B 0,C 180,E1 -23044.693,E2 -23044.693} C_VEL
LIN {X 0,Y 171.858,Z 831.077,A -85,B 0,C 180,E1 -23049.415,E2 -23049.415} C_VEL
LIN {X 0,Y 171.564,Z 831.113,A -85,B 0,C 180,E1 -23054.228,E2 -23054.228} C_VEL
LIN {X 0,Y 171.521,Z 831.121,A -85,B 0,C 180,E1 -23059.87,E2 -23059.87} C_VEL
LIN {X 0,Y 172.173,Z 834.159,A -85,B 0,C 180,E1 -23064.091,E2 -23064.091} C_VEL
LIN {X 0,Y 173.087,Z 838.462,A -85,B 0,C 180,E1 -23069.16,E2 -23069.16} C_VEL
LIN {X 0,Y 174.096,Z 843.422,A -85,B 0,C 180,E1 -23074.413,E2 -23074.413} C_VEL
LIN {X 0,Y 174.87,Z 847.69,A -85,B 0,C 180,E1 -23078.531,E2 -23078.531} C_VEL
LIN {X 0,Y 175.763,Z 852.417,A -85,B 0,C 180,E1 -23082.825,E2 -23082.825} C_VEL
LIN {X 0,Y 176.308,Z 855.248,A -85,B 0,C 180,E1 -23085.171,E2 -23085.171} C_VEL
LIN {X 0,Y 177.598,Z 858.809,A -85,B 0,C 180,E1 -23085.801,E2 -23085.801} C_VEL
LIN {X 0,Y 179.079,Z 861.384,A -85,B 0,C 180,E1 -23086.448,E2 -23086.448} C_VEL
LIN {X 0,Y 180.997,Z 866.903,A -85,B 0,C 180,E1 -23087.475,E2 -23087.475} C_VEL
LIN {X 0,Y 182.525,Z 876.208,A -85,B 0,C 180,E1 -23088.891,E2 -23088.891} C_VEL
LIN {X 0,Y 183.571,Z 888.172,A -85,B 0,C 180,E1 -23090.83,E2 -23090.83} C_VEL
LIN {X 0,Y 183.754,Z 899.989,A -85,B 0,C 180,E1 -23092.981,E2 -23092.981} C_VEL
LIN {X 0,Y 182.989,Z 912.062,A -85,B 0,C 180,E1 -23095.499,E2 -23095.499} C_VEL
LIN {X 0,Y 181.707,Z 922.425,A -85,B 0,C 180,E1 -23098.042,E2 -23098.042} C_VEL
LIN {X 0,Y 179.93,Z 931.88,A -85,B 0,C 180,E1 -23100.78,E2 -23100.78} C_VEL
LIN {X 0,Y 177.98,Z 940.08,A -85,B 0,C 180,E1 -23103.631,E2 -23103.631} C_VEL
LIN {X 0,Y 176.278,Z 945.563,A -85,B 0,C 180,E1 -23105.884,E2 -23105.884} C_VEL
LIN {X 0,Y 173.623,Z 952.42,A -85,B 0,C 180,E1 -23109.261,E2 -23109.261} C_VEL
LIN {X 0,Y 171.625,Z 958.791,A -85,B 0,C 180,E1 -23113.347,E2 -23113.347} C_VEL
LIN {X 0,Y 170.65,Z 962.998,A -85,B 0,C 180,E1 -23116.913,E2 -23116.913} C_VEL
LIN {X 0,Y 170.37,Z 966.177,A -85,B 0,C 180,E1 -23120.507,E2 -23120.507} C_VEL
LIN {X 0,Y 170.465,Z 967.723,A -85,B 0,C 180,E1 -23122.9,E2 -23122.9} C_VEL
LIN {X 0,Y 170.782,Z 968.861,A -85,B 0,C 180,E1 -23125.283,E2 -23125.283} C_VEL
LIN {X 0,Y 171.136,Z 969.576,A -85,B 0,C 180,E1 -23127.651,E2 -23127.651} C_VEL
LIN {X 0,Y 171.509,Z 969.86,A -85,B 0,C 180,E1 -23130.004,E2 -23130.004} C_VEL
LIN {X 0,Y 171.147,Z 969.563,A -85,B 0,C 180,E1 -23132.358,E2 -23132.358} C_VEL
LIN {X 0,Y 170.802,Z 968.839,A -85,B 0,C 180,E1 -23134.725,E2 -23134.725} C_VEL
LIN {X 0,Y 170.4,Z 966.511,A -85,B 0,C 180,E1 -23138.942,E2 -23138.942} C_VEL
LIN {X 0,Y 170.872,Z 962.966,A -85,B 0,C 180,E1 -23143.079,E2 -23143.079} C_VEL
LIN {X 0,Y 171.598,Z 960.422,A -85,B 0,C 180,E1 -23145.348,E2 -23145.348} C_VEL
LIN {X 0,Y 171.918,Z 959.996,A -85,B 0,C 180,E1 -23147.248,E2 -23147.248} C_VEL
LIN {X 0,Y 170.652,Z 958.564,A -85,B 0,C 180,E1 -23150.498,E2 -23150.498} C_VEL
LIN {X 0,Y 169.802,Z 956.875,A -85,B 0,C 180,E1 -23153.822,E2 -23153.822} C_VEL
LIN {X 0,Y 170.804,Z 955.704,A -85,B 0,C 180,E1 -23155.765,E2 -23155.765} C_VEL
LIN {X 0,Y 177.273,Z 951.77,A -85,B 0,C 180,E1 -23161.027,E2 -23161.027} C_VEL
LIN {X 0,Y 185.104,Z 946.202,A -85,B 0,C 180,E1 -23166.055,E2 -23166.055} C_VEL
LIN {X 0,Y 194.527,Z 939.105,A -85,B 0,C 180,E1 -23170.57,E2 -23170.57} C_VEL
LIN {X 0,Y 201.83,Z 932.751,A -85,B 0,C 180,E1 -23174.145,E2 -23174.145} C_VEL
LIN {X 0,Y 209.61,Z 925.654,A -85,B 0,C 180,E1 -23177.888,E2 -23177.888} C_VEL
LIN {X 0,Y 214.124,Z 921.666,A -85,B 0,C 180,E1 -23180.079,E2 -23180.079} C_VEL
LIN {X 0,Y 215.047,Z 920.706,A -85,B 0,C 180,E1 -23180.857,E2 -23180.857} C_VEL
LIN {X 0,Y 215.203,Z 920.058,A -85,B 0,C 180,E1 -23182.415,E2 -23182.415} C_VEL
LIN {X 0,Y 213.308,Z 920.778,A -85,B 0,C 180,E1 -23183.626,E2 -23183.626} C_VEL
LIN {X 0,Y 204.306,Z 924.908,A -85,B 0,C 180,E1 -23186.606,E2 -23186.606} C_VEL
LIN {X 0,Y 195.999,Z 927.524,A -85,B 0,C 180,E1 -23189.867,E2 -23189.867} C_VEL
LIN {X 0,Y 188.56,Z 928.933,A -85,B 0,C 180,E1 -23193.432,E2 -23193.432} C_VEL
LIN {X 0,Y 181.929,Z 929.015,A -85,B 0,C 180,E1 -23197.275,E2 -23197.275} C_VEL
LIN {X 0,Y 176.292,Z 927.744,A -85,B 0,C 180,E1 -23201.402,E2 -23201.402} C_VEL
LIN {X 0,Y 173.848,Z 926.608,A -85,B 0,C 180,E1 -23203.562,E2 -23203.562} C_VEL
LIN {X 0,Y 169.911,Z 923.283,A -85,B 0,C 180,E1 -23208.064,E2 -23208.064} C_VEL
LIN {X 0,Y 167.121,Z 918.447,A -85,B 0,C 180,E1 -23212.752,E2 -23212.752} C_VEL
LIN {X 0,Y 165.653,Z 913.866,A -85,B 0,C 180,E1 -23216.351,E2 -23216.351} C_VEL
LIN {X 0,Y 164.574,Z 908.291,A -85,B 0,C 180,E1 -23220,E2 -23220} C_VEL
LIN {X 0,Y 164.245,Z 901.626,A -85,B 0,C 180,E1 -23223.68,E2 -23223.68} C_VEL
LIN {X 0,Y 164.485,Z 893.795,A -85,B 0,C 180,E1 -23227.365,E2 -23227.365} C_VEL
LIN {X 0,Y 165.136,Z 886.15,A -85,B 0,C 180,E1 -23230.353,E2 -23230.353} C_VEL
LIN {X 0,Y 165.983,Z 876.914,A -85,B 0,C 180,E1 -23233.466,E2 -23233.466} C_VEL
LIN {X 0,Y 166.954,Z 867.355,A -85,B 0,C 180,E1 -23236.194,E2 -23236.194} C_VEL
LIN {X 0,Y 168.096,Z 856.095,A -85,B 0,C 180,E1 -23238.907,E2 -23238.907} C_VEL
LIN {X 0,Y 168.567,Z 850.466,A -85,B 0,C 180,E1 -23240.05,E2 -23240.05} C_VEL
LIN {X 0,Y 166.492,Z 841.475,A -85,B 0,C 180,E1 -23241.762,E2 -23241.762} C_VEL
LIN {X 0,Y 164.5,Z 831.989,A -85,B 0,C 180,E1 -23243.361,E2 -23243.361} C_VEL
LIN {X 0,Y 164.298,Z 832.003,A -85,B 0,C 180,E1 -23248.069,E2 -23248.069} C_VEL
LIN {X 0,Y 164.353,Z 832.002,A -85,B 0,C 180,E1 -23251.208,E2 -23251.208} C_VEL
LIN {X 0,Y 164.288,Z 832.009,A -85,B 0,C 180,E1 -23256.791,E2 -23256.791} C_VEL
LIN {X 0,Y 164.297,Z 832.033,A -85,B 0,C 180,E1 -23262.149,E2 -23262.149} C_VEL
LIN {X 0,Y 165.23,Z 834.773,A -85,B 0,C 180,E1 -23262.887,E2 -23262.887} C_VEL
LIN {X 0,Y 167.265,Z 837.306,A -85,B 0,C 180,E1 -23264.075,E2 -23264.075} C_VEL
LIN {X 0,Y 168.754,Z 840.096,A -85,B 0,C 180,E1 -23265.072,E2 -23265.072} C_VEL
LIN {X 0,Y 171.334,Z 844.338,A -85,B 0,C 180,E1 -23266.727,E2 -23266.727} C_VEL
LIN {X 0,Y 175.778,Z 853.313,A -85,B 0,C 180,E1 -23269.976,E2 -23269.976} C_VEL
LIN {X 0,Y 179.051,Z 861.653,A -85,B 0,C 180,E1 -23272.907,E2 -23272.907} C_VEL
LIN {X 0,Y 181.757,Z 870.908,A -85,B 0,C 180,E1 -23276.199,E2 -23276.199} C_VEL
LIN {X 0,Y 183.353,Z 879.375,A -85,B 0,C 180,E1 -23279.343,E2 -23279.343} C_VEL
LIN {X 0,Y 182.222,Z 883.404,A -85,B 0,C 180,E1 -23280.541,E2 -23280.541} C_VEL
LIN {X 0,Y 179.085,Z 891.437,A -85,B 0,C 180,E1 -23283.169,E2 -23283.169} C_VEL
LIN {X 0,Y 176.301,Z 898.081,A -85,B 0,C 180,E1 -23285.879,E2 -23285.879} C_VEL
LIN {X 0,Y 173.062,Z 905.545,A -85,B 0,C 180,E1 -23289.803,E2 -23289.803} C_VEL
LIN {X 0,Y 170.569,Z 910.538,A -85,B 0,C 180,E1 -23293.232,E2 -23293.232} C_VEL
LIN {X 0,Y 168.378,Z 914.43,A -85,B 0,C 180,E1 -23296.724,E2 -23296.724} C_VEL
LIN {X 0,Y 167.037,Z 917.253,A -85,B 0,C 180,E1 -23300.307,E2 -23300.307} C_VEL
LIN {X 0,Y 166.432,Z 918.596,A -85,B 0,C 180,E1 -23302.718,E2 -23302.718} C_VEL
LIN {X 0,Y 165.5,Z 920.175,A -85,B 0,C 180,E1 -23307.562,E2 -23307.562} C_VEL
LIN {X 0,Y 165.378,Z 920.401,A -85,B 0,C 180,E1 -23309.996,E2 -23309.996} C_VEL
LIN {X 0,Y 165.863,Z 919.627,A -85,B 0,C 180,E1 -23314.857,E2 -23314.857} C_VEL
LIN {X 0,Y 166.4,Z 918.678,A -85,B 0,C 180,E1 -23317.275,E2 -23317.275} C_VEL
LIN {X 0,Y 166.994,Z 917.371,A -85,B 0,C 180,E1 -23319.687,E2 -23319.687} C_VEL
LIN {X 0,Y 168.359,Z 914.58,A -85,B 0,C 180,E1 -23323.268,E2 -23323.268} C_VEL
LIN {X 0,Y 170.556,Z 910.73,A -85,B 0,C 180,E1 -23326.76,E2 -23326.76} C_VEL
LIN {X 0,Y 172.997,Z 905.807,A -85,B 0,C 180,E1 -23330.196,E2 -23330.196} C_VEL
LIN {X 0,Y 175.741,Z 899.617,A -85,B 0,C 180,E1 -23333.568,E2 -23333.568} C_VEL
LIN {X 0,Y 178.372,Z 893.301,A -85,B 0,C 180,E1 -23336.307,E2 -23336.307} C_VEL
LIN {X 0,Y 181.506,Z 885.637,A -85,B 0,C 180,E1 -23338.942,E2 -23338.942} C_VEL
LIN {X 0,Y 183.429,Z 879.765,A -85,B 0,C 180,E1 -23340.676,E2 -23340.676} C_VEL
LIN {X 0,Y 181.972,Z 871.56,A -85,B 0,C 180,E1 -23343.725,E2 -23343.725} C_VEL
LIN {X 0,Y 179.356,Z 862.507,A -85,B 0,C 180,E1 -23346.969,E2 -23346.969} C_VEL
LIN {X 0,Y 176.246,Z 854.25,A -85,B 0,C 180,E1 -23349.859,E2 -23349.859} C_VEL
LIN {X 0,Y 172.351,Z 846.169,A -85,B 0,C 180,E1 -23352.778,E2 -23352.778} C_VEL
LIN {X 0,Y 168.091,Z 838.812,A -85,B 0,C 180,E1 -23355.6,E2 -23355.6} C_VEL
LIN {X 0,Y 167.015,Z 836.686,A -85,B 0,C 180,E1 -23356.329,E2 -23356.329} C_VEL
LIN {X 0,Y 165.067,Z 834.214,A -85,B 0,C 180,E1 -23357.475,E2 -23357.475} C_VEL
LIN {X 0,Y 164.411,Z 831.998,A -85,B 0,C 180,E1 -23358.093,E2 -23358.093} C_VEL
LIN {X 0,Y 164.353,Z 832.013,A -85,B 0,C 180,E1 -23363.226,E2 -23363.226} C_VEL
LIN {X 0,Y 164.379,Z 832.002,A -85,B 0,C 180,E1 -23369.132,E2 -23369.132} C_VEL
LIN {X 0,Y 164.398,Z 831.998,A -85,B 0,C 180,E1 -23374.691,E2 -23374.691} C_VEL
LIN {X 0,Y 164.472,Z 831.99,A -85,B 0,C 180,E1 -23380.049,E2 -23380.049} C_VEL
LIN {X 0,Y 164.522,Z 831.977,A -85,B 0,C 180,E1 -23385.149,E2 -23385.149} C_VEL
LIN {X 0,Y 164.784,Z 831.949,A -85,B 0,C 180,E1 -23390.177,E2 -23390.177} C_VEL
LIN {X 0,Y 164.832,Z 831.951,A -85,B 0,C 180,E1 -23392.651,E2 -23392.651} C_VEL
LIN {X 0,Y 165.035,Z 831.92,A -85,B 0,C 180,E1 -23397.559,E2 -23397.559} C_VEL
LIN {X 0,Y 165.28,Z 831.904,A -85,B 0,C 180,E1 -23400,E2 -23400} C_VEL
LIN {X 0,Y 164.752,Z 831.967,A -85,B 0,C 180,E1 -23404.894,E2 -23404.894} C_VEL
LIN {X 0,Y 164.83,Z 831.954,A -85,B 0,C 180,E1 -23407.349,E2 -23407.349} C_VEL
LIN {X 0,Y 164.735,Z 831.959,A -85,B 0,C 180,E1 -23411.145,E2 -23411.145} C_VEL
LIN {X 0,Y 164.469,Z 832,A -85,B 0,C 180,E1 -23417.405,E2 -23417.405} C_VEL
LIN {X 0,Y 164.509,Z 832.146,A -85,B 0,C 180,E1 -23418.365,E2 -23418.365} C_VEL
LIN {X 0,Y 165.096,Z 835.125,A -85,B 0,C 180,E1 -23422.527,E2 -23422.527} C_VEL
LIN {X 0,Y 165.996,Z 839.237,A -85,B 0,C 180,E1 -23427.757,E2 -23427.757} C_VEL
LIN {X 0,Y 166.987,Z 844.055,A -85,B 0,C 180,E1 -23433.171,E2 -23433.171} C_VEL
LIN {X 0,Y 167.737,Z 847.999,A -85,B 0,C 180,E1 -23437.251,E2 -23437.251} C_VEL
LIN {X 0,Y 168.796,Z 853.697,A -85,B 0,C 180,E1 -23442.578,E2 -23442.578} C_VEL
LIN {X 0,Y 170.095,Z 857.203,A -85,B 0,C 180,E1 -23443.284,E2 -23443.284} C_VEL
LIN {X 0,Y 171.84,Z 860.218,A -85,B 0,C 180,E1 -23444.135,E2 -23444.135} C_VEL
LIN {X 0,Y 173.828,Z 864.763,A -85,B 0,C 180,E1 -23445.192,E2 -23445.192} C_VEL
LIN {X 0,Y 175.859,Z 870.662,A -85,B 0,C 180,E1 -23446.441,E2 -23446.441} C_VEL
LIN {X 0,Y 177.145,Z 881.295,A -85,B 0,C 180,E1 -23448.213,E2 -23448.213} C_VEL
LIN {X 0,Y 177.693,Z 894.003,A -85,B 0,C 180,E1 -23450.524,E2 -23450.524} C_VEL
LIN {X 0,Y 177.227,Z 906.08,A -85,B 0,C 180,E1 -23452.998,E2 -23452.998} C_VEL
LIN {X 0,Y 176.049,Z 917.337,A -85,B 0,C 180,E1 -23455.681,E2 -23455.681} C_VEL
LIN {X 0,Y 174.368,Z 927.062,A -85,B 0,C 180,E1 -23458.406,E2 -23458.406} C_VEL
LIN {X 0,Y 172.289,Z 935.904,A -85,B 0,C 180,E1 -23461.365,E2 -23461.365} C_VEL
LIN {X 0,Y 170.271,Z 943.242,A -85,B 0,C 180,E1 -23464.322,E2 -23464.322} C_VEL
LIN {X 0,Y 167.403,Z 950.332,A -85,B 0,C 180,E1 -23467.805,E2 -23467.805} C_VEL
LIN {X 0,Y 165.258,Z 956.066,A -85,B 0,C 180,E1 -23471.405,E2 -23471.405} C_VEL
LIN {X 0,Y 163.969,Z 960.643,A -85,B 0,C 180,E1 -23475.103,E2 -23475.103} C_VEL
LIN {X 0,Y 163.356,Z 964.153,A -85,B 0,C 180,E1 -23478.842,E2 -23478.842} C_VEL
LIN {X 0,Y 163.399,Z 966.678,A -85,B 0,C 180,E1 -23482.591,E2 -23482.591} C_VEL
LIN {X 0,Y 163.694,Z 967.817,A -85,B 0,C 180,E1 -23485.079,E2 -23485.079} C_VEL
LIN {X 0,Y 164.063,Z 968.537,A -85,B 0,C 180,E1 -23487.549,E2 -23487.549} C_VEL
LIN {X 0,Y 164.464,Z 968.826,A -85,B 0,C 180,E1 -23490.004,E2 -23490.004} C_VEL
LIN {X 0,Y 164.075,Z 968.524,A -85,B 0,C 180,E1 -23492.459,E2 -23492.459} C_VEL
LIN {X 0,Y 163.711,Z 967.794,A -85,B 0,C 180,E1 -23494.93,E2 -23494.93} C_VEL
LIN {X 0,Y 163.376,Z 966.105,A -85,B 0,C 180,E1 -23498.349,E2 -23498.349} C_VEL
LIN {X 0,Y 163.641,Z 963.059,A -85,B 0,C 180,E1 -23502.404,E2 -23502.404} C_VEL
LIN {X 0,Y 165.045,Z 958.722,A -85,B 0,C 180,E1 -23506.709,E2 -23506.709} C_VEL
LIN {X 0,Y 167.676,Z 957.429,A -85,B 0,C 180,E1 -23512.166,E2 -23512.166} C_VEL
LIN {X 0,Y 170.804,Z 955.704,A -85,B 0,C 180,E1 -23515.765,E2 -23515.765} C_VEL
LIN {X 0,Y 172.117,Z 954.57,A -85,B 0,C 180,E1 -23517.656,E2 -23517.656} C_VEL
LIN {X 0,Y 172.993,Z 952.376,A -85,B 0,C 180,E1 -23520.859,E2 -23520.859} C_VEL
LIN {X 0,Y 173.937,Z 950.337,A -85,B 0,C 180,E1 -23523.381,E2 -23523.381} C_VEL
LIN {X 0,Y 175.583,Z 948.632,A -85,B 0,C 180,E1 -23525.162,E2 -23525.162} C_VEL
LIN {X 0,Y 176.405,Z 948.033,A -85,B 0,C 180,E1 -23525.713,E2 -23525.713} C_VEL
LIN {X 0,Y 185.192,Z 942.398,A -85,B 0,C 180,E1 -23530.181,E2 -23530.181} C_VEL
LIN {X 0,Y 191.088,Z 938.301,A -85,B 0,C 180,E1 -23532.879,E2 -23532.879} C_VEL
LIN {X 0,Y 200.655,Z 930.802,A -85,B 0,C 180,E1 -23537.356,E2 -23537.356} C_VEL
LIN {X 0,Y 208.309,Z 924.644,A -85,B 0,C 180,E1 -23540.898,E2 -23540.898} C_VEL
LIN {X 0,Y 208.963,Z 923.841,A -85,B 0,C 180,E1 -23541.898,E2 -23541.898} C_VEL
LIN {X 0,Y 208.137,Z 924.051,A -85,B 0,C 180,E1 -23542.57,E2 -23542.57} C_VEL
LIN {X 0,Y 198.802,Z 927.654,A -85,B 0,C 180,E1 -23545.554,E2 -23545.554} C_VEL
LIN {X 0,Y 190.205,Z 929.849,A -85,B 0,C 180,E1 -23548.849,E2 -23548.849} C_VEL
LIN {X 0,Y 181.606,Z 930.713,A -85,B 0,C 180,E1 -23552.891,E2 -23552.891} C_VEL
LIN {X 0,Y 175.525,Z 930.416,A -85,B 0,C 180,E1 -23556.397,E2 -23556.397} C_VEL
LIN {X 0,Y 169.655,Z 928.732,A -85,B 0,C 180,E1 -23560.646,E2 -23560.646} C_VEL
LIN {X 0,Y 164.834,Z 925.66,A -85,B 0,C 180,E1 -23565.178,E2 -23565.178} C_VEL
LIN {X 0,Y 161.323,Z 921.286,A -85,B 0,C 180,E1 -23569.965,E2 -23569.965} C_VEL
LIN {X 0,Y 159.002,Z 915.296,A -85,B 0,C 180,E1 -23574.928,E2 -23574.928} C_VEL
LIN {X 0,Y 157.723,Z 909.749,A -85,B 0,C 180,E1 -23578.723,E2 -23578.723} C_VEL
LIN {X 0,Y 157.245,Z 903.136,A -85,B 0,C 180,E1 -23582.562,E2 -23582.562} C_VEL
LIN {X 0,Y 157.281,Z 895.361,A -85,B 0,C 180,E1 -23586.414,E2 -23586.414} C_VEL
LIN {X 0,Y 157.949,Z 887.56,A -85,B 0,C 180,E1 -23589.643,E2 -23589.643} C_VEL
LIN {X 0,Y 158.655,Z 878.713,A -85,B 0,C 180,E1 -23592.797,E2 -23592.797} C_VEL
LIN {X 0,Y 159.627,Z 869.331,A -85,B 0,C 180,E1 -23595.645,E2 -23595.645} C_VEL
LIN {X 0,Y 160.773,Z 858.332,A -85,B 0,C 180,E1 -23598.477,E2 -23598.477} C_VEL
LIN {X 0,Y 161.46,Z 851.014,A -85,B 0,C 180,E1 -23600.047,E2 -23600.047} C_VEL
LIN {X 0,Y 158.93,Z 840.21,A -85,B 0,C 180,E1 -23602.142,E2 -23602.142} C_VEL
LIN {X 0,Y 157.45,Z 832.867,A -85,B 0,C 180,E1 -23603.417,E2 -23603.417} C_VEL
LIN {X 0,Y 157.239,Z 832.893,A -85,B 0,C 180,E1 -23609.45,E2 -23609.45} C_VEL
LIN {X 0,Y 157.27,Z 832.877,A -85,B 0,C 180,E1 -23612.429,E2 -23612.429} C_VEL
LIN {X 0,Y 157.267,Z 832.885,A -85,B 0,C 180,E1 -23616.442,E2 -23616.442} C_VEL
LIN {X 0,Y 157.248,Z 832.966,A -85,B 0,C 180,E1 -23619.13,E2 -23619.13} C_VEL
LIN {X 0,Y 158.176,Z 835.583,A -85,B 0,C 180,E1 -23619.944,E2 -23619.944} C_VEL
LIN {X 0,Y 160.11,Z 837.753,A -85,B 0,C 180,E1 -23621.18,E2 -23621.18} C_VEL
LIN {X 0,Y 161.628,Z 840.744,A -85,B 0,C 180,E1 -23622.331,E2 -23622.331} C_VEL
LIN {X 0,Y 165.123,Z 846.312,A -85,B 0,C 180,E1 -23624.803,E2 -23624.803} C_VEL
LIN {X 0,Y 169.692,Z 855.6,A -85,B 0,C 180,E1 -23628.492,E2 -23628.492} C_VEL
LIN {X 0,Y 172.924,Z 863.983,A -85,B 0,C 180,E1 -23631.686,E2 -23631.686} C_VEL
LIN {X 0,Y 175.248,Z 872.072,A -85,B 0,C 180,E1 -23634.762,E2 -23634.762} C_VEL
LIN {X 0,Y 176.791,Z 879.829,A -85,B 0,C 180,E1 -23637.819,E2 -23637.819} C_VEL
LIN {X 0,Y 176.799,Z 882.663,A -85,B 0,C 180,E1 -23638.88,E2 -23638.88} C_VEL
LIN {X 0,Y 173.53,Z 891.008,A -85,B 0,C 180,E1 -23641.579,E2 -23641.579} C_VEL
LIN {X 0,Y 170.429,Z 897.92,A -85,B 0,C 180,E1 -23644.338,E2 -23644.338} C_VEL
LIN {X 0,Y 167.386,Z 904.63,A -85,B 0,C 180,E1 -23647.793,E2 -23647.793} C_VEL
LIN {X 0,Y 164.715,Z 910.007,A -85,B 0,C 180,E1 -23651.332,E2 -23651.332} C_VEL
LIN {X 0,Y 162.189,Z 914.269,A -85,B 0,C 180,E1 -23654.926,E2 -23654.926} C_VEL
LIN {X 0,Y 160.964,Z 916.497,A -85,B 0,C 180,E1 -23657.386,E2 -23657.386} C_VEL
LIN {X 0,Y 160.119,Z 918.285,A -85,B 0,C 180,E1 -23659.884,E2 -23659.884} C_VEL
LIN {X 0,Y 159.468,Z 919.628,A -85,B 0,C 180,E1 -23662.398,E2 -23662.398} C_VEL
LIN {X 0,Y 158.482,Z 921.206,A -85,B 0,C 180,E1 -23667.454,E2 -23667.454} C_VEL
LIN {X 0,Y 158.354,Z 921.432,A -85,B 0,C 180,E1 -23669.995,E2 -23669.995} C_VEL
LIN {X 0,Y 158.865,Z 920.658,A -85,B 0,C 180,E1 -23675.071,E2 -23675.071} C_VEL
LIN {X 0,Y 159.438,Z 919.709,A -85,B 0,C 180,E1 -23677.594,E2 -23677.594} C_VEL
LIN {X 0,Y 160.081,Z 918.401,A -85,B 0,C 180,E1 -23680.11,E2 -23680.11} C_VEL
LIN {X 0,Y 161.53,Z 915.61,A -85,B 0,C 180,E1 -23683.84,E2 -23683.84} C_VEL
LIN {X 0,Y 163.842,Z 911.76,A -85,B 0,C 180,E1 -23687.469,E2 -23687.469} C_VEL
LIN {X 0,Y 166.425,Z 906.836,A -85,B 0,C 180,E1 -23691.031,E2 -23691.031} C_VEL
LIN {X 0,Y 169.323,Z 900.646,A -85,B 0,C 180,E1 -23694.518,E2 -23694.518} C_VEL
LIN {X 0,Y 172.103,Z 894.33,A -85,B 0,C 180,E1 -23697.344,E2 -23697.344} C_VEL
LIN {X 0,Y 175.392,Z 886.665,A -85,B 0,C 180,E1 -23700.053,E2 -23700.053} C_VEL
LIN {X 0,Y 177.063,Z 881.576,A -85,B 0,C 180,E1 -23701.637,E2 -23701.637} C_VEL
LIN {X 0,Y 175.828,Z 874.223,A -85,B 0,C 180,E1 -23704.566,E2 -23704.566} C_VEL
LIN {X 0,Y 173.553,Z 865.822,A -85,B 0,C 180,E1 -23707.801,E2 -23707.801} C_VEL
LIN {X 0,Y 170.571,Z 857.544,A -85,B 0,C 180,E1 -23710.948,E2 -23710.948} C_VEL
LIN {X 0,Y 167.467,Z 850.681,A -85,B 0,C 180,E1 -23713.62,E2 -23713.62} C_VEL
LIN {X 0,Y 163.566,Z 843.521,A -85,B 0,C 180,E1 -23716.569,E2 -23716.569} C_VEL
LIN {X 0,Y 160.645,Z 838.602,A -85,B 0,C 180,E1 -23718.674,E2 -23718.674} C_VEL
LIN {X 0,Y 159.971,Z 837.574,A -85,B 0,C 180,E1 -23719.145,E2 -23719.145} C_VEL
LIN {X 0,Y 157.985,Z 835.133,A -85,B 0,C 180,E1 -23720.448,E2 -23720.448} C_VEL
LIN {X 0,Y 157.293,Z 832.883,A -85,B 0,C 180,E1 -23721.175,E2 -23721.175} C_VEL
LIN {X 0,Y 157.305,Z 832.884,A -85,B 0,C 180,E1 -23724.492,E2 -23724.492} C_VEL
LIN {X 0,Y 157.286,Z 832.893,A -85,B 0,C 180,E1 -23728.09,E2 -23728.09} C_VEL
LIN {X 0,Y 157.306,Z 832.884,A -85,B 0,C 180,E1 -23733.463,E2 -23733.463} C_VEL
LIN {X 0,Y 157.381,Z 832.872,A -85,B 0,C 180,E1 -23739.666,E2 -23739.666} C_VEL
LIN {X 0,Y 157.448,Z 832.857,A -85,B 0,C 180,E1 -23744.465,E2 -23744.465} C_VEL
LIN {X 0,Y 157.712,Z 832.832,A -85,B 0,C 180,E1 -23749.732,E2 -23749.732} C_VEL
LIN {X 0,Y 157.789,Z 832.825,A -85,B 0,C 180,E1 -23752.321,E2 -23752.321} C_VEL
LIN {X 0,Y 158.243,Z 832.781,A -85,B 0,C 180,E1 -23760,E2 -23760} C_VEL
LIN {X 0,Y 157.787,Z 832.833,A -85,B 0,C 180,E1 -23767.679,E2 -23767.679} C_VEL
LIN {X 0,Y 157.676,Z 832.836,A -85,B 0,C 180,E1 -23771.335,E2 -23771.335} C_VEL
LIN {X 0,Y 157.447,Z 833.067,A -85,B 0,C 180,E1 -23776.199,E2 -23776.199} C_VEL
LIN {X 0,Y 158.076,Z 836.19,A -85,B 0,C 180,E1 -23781.003,E2 -23781.003} C_VEL
LIN {X 0,Y 158.914,Z 840.045,A -85,B 0,C 180,E1 -23786.248,E2 -23786.248} C_VEL
LIN {X 0,Y 159.647,Z 843.449,A -85,B 0,C 180,E1 -23790.415,E2 -23790.415} C_VEL
LIN {X 0,Y 160.684,Z 848.641,A -85,B 0,C 180,E1 -23796.19,E2 -23796.19} C_VEL
LIN {X 0,Y 161.262,Z 852.007,A -85,B 0,C 180,E1 -23799.575,E2 -23799.575} C_VEL
LIN {X 0,Y 162.716,Z 855.811,A -85,B 0,C 180,E1 -23800.469,E2 -23800.469} C_VEL
LIN {X 0,Y 164.652,Z 859.086,A -85,B 0,C 180,E1 -23801.533,E2 -23801.533} C_VEL
LIN {X 0,Y 166.685,Z 863.55,A -85,B 0,C 180,E1 -23802.732,E2 -23802.732} C_VEL
LIN {X 0,Y 169.81,Z 871.295,A -85,B 0,C 180,E1 -23804.715,E2 -23804.715} C_VEL
LIN {X 0,Y 170.624,Z 874.271,A -85,B 0,C 180,E1 -23805.361,E2 -23805.361} C_VEL
LIN {X 0,Y 171.61,Z 887.066,A -85,B 0,C 180,E1 -23807.719,E2 -23807.719} C_VEL
LIN {X 0,Y 171.546,Z 899.151,A -85,B 0,C 180,E1 -23810.167,E2 -23810.167} C_VEL
LIN {X 0,Y 170.505,Z 911.196,A -85,B 0,C 180,E1 -23812.933,E2 -23812.933} C_VEL
LIN {X 0,Y 168.847,Z 922.059,A -85,B 0,C 180,E1 -23815.88,E2 -23815.88} C_VEL
LIN {X 0,Y 166.753,Z 931.469,A -85,B 0,C 180,E1 -23818.922,E2 -23818.922} C_VEL
LIN {X 0,Y 164.159,Z 940.797,A -85,B 0,C 180,E1 -23822.603,E2 -23822.603} C_VEL
LIN {X 0,Y 161.805,Z 947.015,A -85,B 0,C 180,E1 -23825.596,E2 -23825.596} C_VEL
LIN {X 0,Y 159.11,Z 953.24,A -85,B 0,C 180,E1 -23829.312,E2 -23829.312} C_VEL
LIN {X 0,Y 157.451,Z 958.199,A -85,B 0,C 180,E1 -23833.139,E2 -23833.139} C_VEL
LIN {X 0,Y 156.487,Z 962.05,A -85,B 0,C 180,E1 -23837.028,E2 -23837.028} C_VEL
LIN {X 0,Y 156.327,Z 965.251,A -85,B 0,C 180,E1 -23841.515,E2 -23841.515} C_VEL
LIN {X 0,Y 156.611,Z 966.774,A -85,B 0,C 180,E1 -23844.855,E2 -23844.855} C_VEL
LIN {X 0,Y 156.987,Z 967.497,A -85,B 0,C 180,E1 -23847.439,E2 -23847.439} C_VEL
LIN {X 0,Y 157.416,Z 967.791,A -85,B 0,C 180,E1 -23850.005,E2 -23850.005} C_VEL
LIN {X 0,Y 156.999,Z 967.484,A -85,B 0,C 180,E1 -23852.57,E2 -23852.57} C_VEL
LIN {X 0,Y 156.626,Z 966.75,A -85,B 0,C 180,E1 -23855.153,E2 -23855.153} C_VEL
LIN {X 0,Y 156.334,Z 965.2,A -85,B 0,C 180,E1 -23858.501,E2 -23858.501} C_VEL
LIN {X 0,Y 156.686,Z 962.011,A -85,B 0,C 180,E1 -23862.964,E2 -23862.964} C_VEL
LIN {X 0,Y 158.502,Z 957.033,A -85,B 0,C 180,E1 -23867.92,E2 -23867.92} C_VEL
LIN {X 0,Y 161.157,Z 956.157,A -85,B 0,C 180,E1 -23873.114,E2 -23873.114} C_VEL
LIN {X 0,Y 165.511,Z 954.224,A -85,B 0,C 180,E1 -23877.85,E2 -23877.85} C_VEL
LIN {X 0,Y 171.198,Z 951.185,A -85,B 0,C 180,E1 -23882.259,E2 -23882.259} C_VEL
LIN {X 0,Y 176.405,Z 948.033,A -85,B 0,C 180,E1 -23885.713,E2 -23885.713} C_VEL
LIN {X 0,Y 178.638,Z 946.259,A -85,B 0,C 180,E1 -23887.383,E2 -23887.383} C_VEL
LIN {X 0,Y 181.164,Z 943.39,A -85,B 0,C 180,E1 -23890.292,E2 -23890.292} C_VEL
LIN {X 0,Y 183.278,Z 940.99,A -85,B 0,C 180,E1 -23892.589,E2 -23892.589} C_VEL
LIN {X 0,Y 186.536,Z 938.354,A -85,B 0,C 180,E1 -23894.675,E2 -23894.675} C_VEL
LIN {X 0,Y 195.9,Z 931.979,A -85,B 0,C 180,E1 -23898.889,E2 -23898.889} C_VEL
LIN {X 0,Y 200.324,Z 928.876,A -85,B 0,C 180,E1 -23900.839,E2 -23900.839} C_VEL
LIN {X 0,Y 201.778,Z 927.704,A -85,B 0,C 180,E1 -23901.812,E2 -23901.812} C_VEL
LIN {X 0,Y 193.323,Z 930.232,A -85,B 0,C 180,E1 -23904.433,E2 -23904.433} C_VEL
LIN {X 0,Y 188.781,Z 931.296,A -85,B 0,C 180,E1 -23906.053,E2 -23906.053} C_VEL
LIN {X 0,Y 180.301,Z 932.395,A -85,B 0,C 180,E1 -23909.554,E2 -23909.554} C_VEL
LIN {X 0,Y 172.653,Z 932.219,A -85,B 0,C 180,E1 -23913.4,E2 -23913.4} C_VEL
LIN {X 0,Y 165.967,Z 930.786,A -85,B 0,C 180,E1 -23917.598,E2 -23917.598} C_VEL
LIN {X 0,Y 163.023,Z 929.583,A -85,B 0,C 180,E1 -23919.825,E2 -23919.825} C_VEL
LIN {X 0,Y 158.003,Z 926.125,A -85,B 0,C 180,E1 -23924.521,E2 -23924.521} C_VEL
LIN {X 0,Y 154.36,Z 921.24,A -85,B 0,C 180,E1 -23929.507,E2 -23929.507} C_VEL
LIN {X 0,Y 152.487,Z 916.662,A -85,B 0,C 180,E1 -23933.384,E2 -23933.384} C_VEL
LIN {X 0,Y 150.985,Z 911.13,A -85,B 0,C 180,E1 -23937.332,E2 -23937.332} C_VEL
LIN {X 0,Y 150.321,Z 904.56,A -85,B 0,C 180,E1 -23941.34,E2 -23941.34} C_VEL
LIN {X 0,Y 150.177,Z 896.84,A -85,B 0,C 180,E1 -23945.371,E2 -23945.371} C_VEL
LIN {X 0,Y 150.827,Z 887.554,A -85,B 0,C 180,E1 -23949.386,E2 -23949.386} C_VEL
LIN {X 0,Y 151.617,Z 877.976,A -85,B 0,C 180,E1 -23952.893,E2 -23952.893} C_VEL
LIN {X 0,Y 152.804,Z 866.674,A -85,B 0,C 180,E1 -23956.363,E2 -23956.363} C_VEL
LIN {X 0,Y 154.004,Z 854.782,A -85,B 0,C 180,E1 -23959.321,E2 -23959.321} C_VEL
LIN {X 0,Y 154.331,Z 851.74,A -85,B 0,C 180,E1 -23959.971,E2 -23959.971} C_VEL
LIN {X 0,Y 152.122,Z 842.212,A -85,B 0,C 180,E1 -23961.903,E2 -23961.903} C_VEL
LIN {X 0,Y 150.41,Z 833.744,A -85,B 0,C 180,E1 -23963.491,E2 -23963.491} C_VEL
LIN {X 0,Y 150.168,Z 833.762,A -85,B 0,C 180,E1 -23967.905,E2 -23967.905} C_VEL
LIN {X 0,Y 150.211,Z 833.756,A -85,B 0,C 180,E1 -23972.622,E2 -23972.622} C_VEL
LIN {X 0,Y 150.242,Z 833.818,A -85,B 0,C 180,E1 -23975.577,E2 -23975.577} C_VEL
LIN {X 0,Y 151.101,Z 836.374,A -85,B 0,C 180,E1 -23976.478,E2 -23976.478} C_VEL
LIN {X 0,Y 153.039,Z 838.642,A -85,B 0,C 180,E1 -23977.915,E2 -23977.915} C_VEL
LIN {X 0,Y 153.662,Z 839.498,A -85,B 0,C 180,E1 -23978.396,E2 -23978.396} C_VEL
LIN {X 0,Y 155.116,Z 842.215,A -85,B 0,C 180,E1 -23979.619,E2 -23979.619} C_VEL
LIN {X 0,Y 156.468,Z 844.007,A -85,B 0,C 180,E1 -23980.638,E2 -23980.638} C_VEL
LIN {X 0,Y 160.91,Z 852.021,A -85,B 0,C 180,E1 -23984.333,E2 -23984.333} C_VEL
LIN {X 0,Y 165.128,Z 861.425,A -85,B 0,C 180,E1 -23988.362,E2 -23988.362} C_VEL
LIN {X 0,Y 167.844,Z 869.571,A -85,B 0,C 180,E1 -23991.7,E2 -23991.7} C_VEL
LIN {X 0,Y 169.527,Z 876.431,A -85,B 0,C 180,E1 -23994.517,E2 -23994.517} C_VEL
LIN {X 0,Y 170.701,Z 883.719,A -85,B 0,C 180,E1 -23997.636,E2 -23997.636} C_VEL
LIN {X 0,Y 168.068,Z 890.47,A -85,B 0,C 180,E1 -23999.877,E2 -23999.877} C_VEL
LIN {X 0,Y 164.685,Z 897.655,A -85,B 0,C 180,E1 -24002.688,E2 -24002.688} C_VEL
LIN {X 0,Y 161.872,Z 903.751,A -85,B 0,C 180,E1 -24005.75,E2 -24005.75} C_VEL
LIN {X 0,Y 159.038,Z 909.373,A -85,B 0,C 180,E1 -24009.292,E2 -24009.292} C_VEL
LIN {X 0,Y 156.232,Z 914.009,A -85,B 0,C 180,E1 -24012.994,E2 -24012.994} C_VEL
LIN {X 0,Y 154.116,Z 917.529,A -85,B 0,C 180,E1 -24016.815,E2 -24016.815} C_VEL
LIN {X 0,Y 153.21,Z 919.316,A -85,B 0,C 180,E1 -24019.422,E2 -24019.422} C_VEL
LIN {X 0,Y 152.509,Z 920.659,A -85,B 0,C 180,E1 -24022.049,E2 -24022.049} C_VEL
LIN {X 0,Y 151.466,Z 922.237,A -85,B 0,C 180,E1 -24027.336,E2 -24027.336} C_VEL
LIN {X 0,Y 151.33,Z 922.464,A -85,B 0,C 180,E1 -24029.995,E2 -24029.995} C_VEL
LIN {X 0,Y 151.87,Z 921.688,A -85,B 0,C 180,E1 -24035.306,E2 -24035.306} C_VEL
LIN {X 0,Y 152.481,Z 920.739,A -85,B 0,C 180,E1 -24037.943,E2 -24037.943} C_VEL
LIN {X 0,Y 153.175,Z 919.43,A -85,B 0,C 180,E1 -24040.57,E2 -24040.57} C_VEL
LIN {X 0,Y 154.718,Z 916.641,A -85,B 0,C 180,E1 -24044.463,E2 -24044.463} C_VEL
LIN {X 0,Y 157.155,Z 912.79,A -85,B 0,C 180,E1 -24048.238,E2 -24048.238} C_VEL
LIN {X 0,Y 159.894,Z 907.865,A -85,B 0,C 180,E1 -24051.933,E2 -24051.933} C_VEL
LIN {X 0,Y 162.958,Z 901.676,A -85,B 0,C 180,E1 -24055.543,E2 -24055.543} C_VEL
LIN {X 0,Y 165.895,Z 895.359,A -85,B 0,C 180,E1 -24058.458,E2 -24058.458} C_VEL
LIN {X 0,Y 169.35,Z 887.693,A -85,B 0,C 180,E1 -24061.243,E2 -24061.243} C_VEL
LIN {X 0,Y 170.704,Z 884.212,A -85,B 0,C 180,E1 -24062.353,E2 -24062.353} C_VEL
LIN {X 0,Y 169.704,Z 876.958,A -85,B 0,C 180,E1 -24065.43,E2 -24065.43} C_VEL
LIN {X 0,Y 167.548,Z 868.382,A -85,B 0,C 180,E1 -24068.984,E2 -24068.984} C_VEL
LIN {X 0,Y 164.544,Z 859.719,A -85,B 0,C 180,E1 -24072.542,E2 -24072.542} C_VEL
LIN {X 0,Y 161.124,Z 852.27,A -85,B 0,C 180,E1 -24075.741,E2 -24075.741} C_VEL
LIN {X 0,Y 156.114,Z 843.248,A -85,B 0,C 180,E1 -24079.927,E2 -24079.927} C_VEL
LIN {X 0,Y 154.036,Z 840.224,A -85,B 0,C 180,E1 -24081.531,E2 -24081.531} C_VEL
LIN {X 0,Y 153.387,Z 838.799,A -85,B 0,C 180,E1 -24082.129,E2 -24082.129} C_VEL
LIN {X 0,Y 151.253,Z 836.568,A -85,B 0,C 180,E1 -24083.67,E2 -24083.67} C_VEL
LIN {X 0,Y 150.286,Z 833.989,A -85,B 0,C 180,E1 -24084.64,E2 -24084.64} C_VEL
LIN {X 0,Y 150.22,Z 833.764,A -85,B 0,C 180,E1 -24085.032,E2 -24085.032} C_VEL
LIN {X 0,Y 150.197,Z 833.768,A -85,B 0,C 180,E1 -24089.022,E2 -24089.022} C_VEL
LIN {X 0,Y 150.23,Z 833.771,A -85,B 0,C 180,E1 -24092.717,E2 -24092.717} C_VEL
LIN {X 0,Y 150.338,Z 833.749,A -85,B 0,C 180,E1 -24099.206,E2 -24099.206} C_VEL
LIN {X 0,Y 150.354,Z 833.743,A -85,B 0,C 180,E1 -24103.712,E2 -24103.712} C_VEL
LIN {X 0,Y 150.639,Z 833.716,A -85,B 0,C 180,E1 -24109.244,E2 -24109.244} C_VEL
LIN {X 0,Y 150.725,Z 833.702,A -85,B 0,C 180,E1 -24111.959,E2 -24111.959} C_VEL
LIN {X 0,Y 151.203,Z 833.658,A -85,B 0,C 180,E1 -24120,E2 -24120} C_VEL
LIN {X 0,Y 150.723,Z 833.711,A -85,B 0,C 180,E1 -24128.041,E2 -24128.041} C_VEL
LIN {X 0,Y 150.509,Z 833.725,A -85,B 0,C 180,E1 -24132.819,E2 -24132.819} C_VEL
LIN {X 0,Y 150.44,Z 833.804,A -85,B 0,C 180,E1 -24133.508,E2 -24133.508} C_VEL
LIN {X 0,Y 151.092,Z 837.051,A -85,B 0,C 180,E1 -24139.002,E2 -24139.002} C_VEL
LIN {X 0,Y 151.856,Z 840.89,A -85,B 0,C 180,E1 -24144.615,E2 -24144.615} C_VEL
LIN {X 0,Y 152.81,Z 845.306,A -85,B 0,C 180,E1 -24150.392,E2 -24150.392} C_VEL
LIN {X 0,Y 153.773,Z 850.24,A -85,B 0,C 180,E1 -24156.066,E2 -24156.066} C_VEL
LIN {X 0,Y 155.185,Z 853.94,A -85,B 0,C 180,E1 -24157.078,E2 -24157.078} C_VEL
LIN {X 0,Y 157.35,Z 857.439,A -85,B 0,C 180,E1 -24158.434,E2 -24158.434} C_VEL
LIN {X 0,Y 159.227,Z 861.787,A -85,B 0,C 180,E1 -24159.725,E2 -24159.725} C_VEL
LIN {X 0,Y 160.381,Z 864.046,A -85,B 0,C 180,E1 -24160.473,E2 -24160.473} C_VEL
LIN {X 0,Y 163.025,Z 870.505,A -85,B 0,C 180,E1 -24162.345,E2 -24162.345} C_VEL
LIN {X 0,Y 165.191,Z 876.667,A -85,B 0,C 180,E1 -24164.033,E2 -24164.033} C_VEL
LIN {X 0,Y 165.827,Z 889.217,A -85,B 0,C 180,E1 -24166.534,E2 -24166.534} C_VEL
LIN {X 0,Y 165.407,Z 901.469,A -85,B 0,C 180,E1 -24169.219,E2 -24169.219} C_VEL
LIN {X 0,Y 164.119,Z 912.642,A -85,B 0,C 180,E1 -24172.012,E2 -24172.012} C_VEL
LIN {X 0,Y 162.202,Z 923.225,A -85,B 0,C 180,E1 -24175.113,E2 -24175.113} C_VEL
LIN {X 0,Y 159.993,Z 932.093,A -85,B 0,C 180,E1 -24178.195,E2 -24178.195} C_VEL
LIN {X 0,Y 157.707,Z 939.726,A -85,B 0,C 180,E1 -24181.382,E2 -24181.382} C_VEL
LIN {X 0,Y 155.737,Z 944.991,A -85,B 0,C 180,E1 -24183.974,E2 -24183.974} C_VEL
LIN {X 0,Y 152.441,Z 952.191,A -85,B 0,C 180,E1 -24188.362,E2 -24188.362} C_VEL
LIN {X 0,Y 150.613,Z 957.149,A -85,B 0,C 180,E1 -24192.349,E2 -24192.349} C_VEL
LIN {X 0,Y 149.523,Z 961.001,A -85,B 0,C 180,E1 -24196.413,E2 -24196.413} C_VEL
LIN {X 0,Y 149.262,Z 964.362,A -85,B 0,C 180,E1 -24201.411,E2 -24201.411} C_VEL
LIN {X 0,Y 149.533,Z 965.73,A -85,B 0,C 180,E1 -24204.611,E2 -24204.611} C_VEL
LIN {X 0,Y 149.908,Z 966.457,A -85,B 0,C 180,E1 -24207.318,E2 -24207.318} C_VEL
LIN {X 0,Y 150.364,Z 966.756,A -85,B 0,C 180,E1 -24210.005,E2 -24210.005} C_VEL
LIN {X 0,Y 149.92,Z 966.443,A -85,B 0,C 180,E1 -24212.692,E2 -24212.692} C_VEL
LIN {X 0,Y 149.546,Z 965.706,A -85,B 0,C 180,E1 -24215.398,E2 -24215.398} C_VEL
LIN {X 0,Y 149.293,Z 964.288,A -85,B 0,C 180,E1 -24218.667,E2 -24218.667} C_VEL
LIN {X 0,Y 149.753,Z 960.965,A -85,B 0,C 180,E1 -24223.576,E2 -24223.576} C_VEL
LIN {X 0,Y 151.147,Z 957.141,A -85,B 0,C 180,E1 -24227.597,E2 -24227.597} C_VEL
LIN {X 0,Y 151.997,Z 955.327,A -85,B 0,C 180,E1 -24229.24,E2 -24229.24} C_VEL
LIN {X 0,Y 155.955,Z 954.357,A -85,B 0,C 180,E1 -24235.672,E2 -24235.672} C_VEL
LIN {X 0,Y 162.114,Z 952.011,A -85,B 0,C 180,E1 -24241.352,E2 -24241.352} C_VEL
LIN {X 0,Y 168.394,Z 948.839,A -85,B 0,C 180,E1 -24245.758,E2 -24245.758} C_VEL
LIN {X 0,Y 175.724,Z 944.881,A -85,B 0,C 180,E1 -24249.79,E2 -24249.79} C_VEL
LIN {X 0,Y 183.921,Z 940.109,A -85,B 0,C 180,E1 -24253.462,E2 -24253.462} C_VEL
LIN {X 0,Y 186.536,Z 938.354,A -85,B 0,C 180,E1 -24254.675,E2 -24254.675} C_VEL
LIN {X 0,Y 188.138,Z 937.079,A -85,B 0,C 180,E1 -24255.704,E2 -24255.704} C_VEL
LIN {X 0,Y 189.459,Z 935.328,A -85,B 0,C 180,E1 -24257.605,E2 -24257.605} C_VEL
LIN {X 0,Y 190.731,Z 933.41,A -85,B 0,C 180,E1 -24259.967,E2 -24259.967} C_VEL
LIN {X 0,Y 191.517,Z 932.705,A -85,B 0,C 180,E1 -24260.717,E2 -24260.717} C_VEL
LIN {X 0,Y 192.844,Z 931.687,A -85,B 0,C 180,E1 -24261.717,E2 -24261.717} C_VEL
LIN {X 0,Y 183.207,Z 933.507,A -85,B 0,C 180,E1 -24264.871,E2 -24264.871} C_VEL
LIN {X 0,Y 174.377,Z 934.108,A -85,B 0,C 180,E1 -24268.403,E2 -24268.403} C_VEL
LIN {X 0,Y 167.77,Z 933.766,A -85,B 0,C 180,E1 -24271.614,E2 -24271.614} C_VEL
LIN {X 0,Y 162.795,Z 932.801,A -85,B 0,C 180,E1 -24274.424,E2 -24274.424} C_VEL
LIN {X 0,Y 156.403,Z 930.209,A -85,B 0,C 180,E1 -24278.932,E2 -24278.932} C_VEL
LIN {X 0,Y 152.383,Z 927.479,A -85,B 0,C 180,E1 -24282.555,E2 -24282.555} C_VEL
LIN {X 0,Y 148.24,Z 922.555,A -85,B 0,C 180,E1 -24287.682,E2 -24287.682} C_VEL
LIN {X 0,Y 146.057,Z 917.958,A -85,B 0,C 180,E1 -24291.7,E2 -24291.7} C_VEL
